# B&R Automation Studio project OpcUaSample410_BrbLibUa103 (part 4)

#### BrbReadDir.c - Gibt eine Liste der Dateien eines Laufwerks zurück
```c
/********************************************************************
 * COPYRIGHT -- Bernecker + Rainer
 ********************************************************************
 * Library: BrbLib
 * File: BrbReadDir.c
 * Author: niedermeierr
 * Created: June 17, 2013
 ********************************************************************
 * Implementation of library BrbLib
 ********************************************************************/

#include <bur/plctypes.h>
#ifdef __cplusplus
	extern "C"
	{
#endif

#include "BrbLib.h"
#include <string.h>
#include <AnsiCFunc.h>

#ifdef __cplusplus
	};
#endif

// NOLINTBEGIN(readability-*, bugprone-easily-swappable-parameters, clang-diagnostic-invalid-utf8, clang-diagnostic-invalid-source-encoding, clang-diagnostic-pointer-arith, clang-diagnostic-strict-prototypes, hicpp-uppercase-literal-suffix, cppcoreguidelines-*, performance-*)

// Eigene Enums und Typen
enum Steps_ENUM
{
	eSTEP_INIT,
	eSTEP_GET_FILTER,
	eSTEP_READ_DIR,
	eSTEP_SORT,
};

// Prototypen
BOOL CallUserFilterFunction(struct BrbReadDir* inst, fiDIR_READ_DATA* pFileInfo);
void SortList(struct BrbReadDir* inst);
INT SortTwoEntries(fiDIR_READ_DATA* pEntry1, fiDIR_READ_DATA* pEntry2, BrbFileSorting_ENUM eSorting, BOOL bCaseSensitive, UDINT pUserCompareFunction);
INT FileComparerNone(fiDIR_READ_DATA* pEntry1, fiDIR_READ_DATA* pEntry2);
INT FileComparerAlphUp(fiDIR_READ_DATA* pEntry1, fiDIR_READ_DATA* pEntry2);
INT FileComparerAlphUpCaseSensitive(fiDIR_READ_DATA* pEntry1, fiDIR_READ_DATA* pEntry2);
INT FileComparerAlphDown(fiDIR_READ_DATA* pEntry1, fiDIR_READ_DATA* pEntry2);
INT FileComparerAlphDownCaseSensitive(fiDIR_READ_DATA* pEntry1, fiDIR_READ_DATA* pEntry2);
INT FileComparerOldest(fiDIR_READ_DATA* pEntry1, fiDIR_READ_DATA* pEntry2);
INT FileComparerYoungest(fiDIR_READ_DATA* pEntry1, fiDIR_READ_DATA* pEntry2);
INT FileComparerBiggest(fiDIR_READ_DATA* pEntry1, fiDIR_READ_DATA* pEntry2);
INT FileComparerSmallest(fiDIR_READ_DATA* pEntry1, fiDIR_READ_DATA* pEntry2);

/* Gibt eine Liste der Dateien und/oder der Verzeichnisse eines Laufwerks zurück */
void BrbReadDir(struct BrbReadDir* inst) // NOLINT(readability-function-cognitive-complexity)
{
	// Prüfung der Parameter
	if(inst->pDevice == 0)
	{
		inst->nStatus = eBRB_ERR_NULL_POINTER;
		return;
	}
	if(inst->pFileFilter == 0)
	{
		inst->nStatus = eBRB_ERR_NULL_POINTER;
		return;
	}

	if(inst->pList == 0)
	{
		inst->nStatus = eBRB_ERR_NULL_POINTER;
		return;
	}

	switch(inst->eStep)
	{
		case eSTEP_INIT:
			// Fub initialisieren
			inst->nStatus = eBRB_ERR_BUSY;
			inst->nDirCount = 0;
			inst->nFileCount = 0;
			inst->nTotalCount = 0;
			memset(&inst->FilterListMan, 0, sizeof(inst->FilterListMan));
			memset(&inst->fbDirRead, 0, sizeof(inst->fbDirRead));
			memset(&inst->FileInfo, 0, sizeof(inst->FileInfo));
			memset(&inst->FileListMan, 0, sizeof(inst->FileListMan));
			// Der Einfachkeit halber wird das File-Array in einer MemList verwaltet
			inst->FileListMan.pList = inst->pList;
			inst->FileListMan.nIndexMax = inst->nListIndexMax;
			inst->FileListMan.nEntryLength = sizeof(inst->ReadListEntry);
			BrbMemListClear(&inst->FileListMan);
			// Prüfen, ob bei benutzerdefinierter Filterung eine Funktion angegeben ist
			inst->eStep = eSTEP_GET_FILTER;
			if(inst->bUserFilter == 1)
			{
				if(inst->pUserFilterFunction == 0)
				{
					inst->nStatus = fiERR_PARAMETER;
					inst->eStep = eSTEP_INIT;
				}
			}
			// Prüfen, ob bei benutzerdefinierter Sortierung eine Vergleichsfunktion angegeben ist
			if(inst->eSorting == eBRB_FILE_SORTING_USER)
			{
				if(inst->pUserCompareFunction == 0)
				{
					inst->nStatus = fiERR_PARAMETER;
					inst->eStep = eSTEP_INIT;
				}
			}
			break;

		case eSTEP_GET_FILTER:
			// Filtertext in Liste umsetzen
			// Der Einfachkeit halber wird die Filter-Liste in einer MemList verwaltet
			inst->FilterListMan.pList = (UDINT)&inst->FilterList;
			inst->FilterListMan.nIndexMax = nBRB_FILTER_SINGLE_INDEX_MAX;
			inst->FilterListMan.nEntryLength = nBRB_FILTER_SINGLE_CHAR_MAX+1;
			BrbMemListClear(&inst->FilterListMan);
			if(strlen(inst->pFileFilter))
			{
				inst->FilterListMan.nEntryCount = BrbStringSplit(inst->pFileFilter, ";", inst->FilterListMan.pList, inst->FilterListMan.nIndexMax, inst->FilterListMan.nEntryLength);
			}
			inst->eStep = eSTEP_READ_DIR;
			break;

		case eSTEP_READ_DIR:
			// Laufwerk auslesen
			inst->nStatus = eBRB_ERR_BUSY;
			inst->fbDirRead.enable = 1;
			inst->fbDirRead.pDevice = (UDINT)inst->pDevice;
			inst->fbDirRead.pPath = (UDINT)inst->pPath;
			inst->fbDirRead.option = fiBOTH;
			inst->fbDirRead.pData = (UDINT)&inst->FileInfo;
			inst->fbDirRead.data_len = sizeof(inst->FileInfo);
			DirRead(&inst->fbDirRead);
			if(inst->fbDirRead.status == 0)
			{
				// Filterprüfung
				BOOL bInFilter = 0;
				// Interner Filter (Dateiendung)
				if((strcmp((STRING*)&inst->FileInfo.Filename, "..") == 0 && inst->bWithParentDir == 0) || strcmp((STRING*)&inst->FileInfo.Filename, ".") == 0)
				{
					// ".." bezieht sich auf das übergeordnete Verzeichnis und wird nur optional zurückgegeben
					// "." bezieht sich auf das eigene Verzeichnis und wird grundsätzlich nicht zurückgegeben
				}
				else if(strcmp((STRING*)&inst->FileInfo.Filename, "..") == 0 && inst->bWithParentDir == 1)
				{
					// ".." bezieht sich auf das übergeordnete Verzeichnis und wird nur optional zurückgegeben
					bInFilter = 1;
					inst->nDirCount += 1;
				}
				else if(inst->eFilter != eBRB_DIR_INFO_ONLY_FILES && inst->FileInfo.Filelength == 0)
				{
					// Verzeichnis
					BOOL bInUserFilter = CallUserFilterFunction(inst, &inst->FileInfo);
					if(bInUserFilter == 1)
					{
						bInFilter = 1;
						inst->nDirCount += 1;
					}
				}
				else if(inst->eFilter != eBRB_DIR_INFO_ONLY_DIRS && inst->FileInfo.Filelength > 0)
				{
					if(inst->FilterListMan.nEntryCount > 0)
					{
						UDINT nFilterListIndex = 0;
						for(nFilterListIndex=0; nFilterListIndex<inst->FilterListMan.nEntryCount; nFilterListIndex++)
						{
							if(BrbStringEndsWith((STRING*)&inst->FileInfo.Filename, inst->FilterList[nFilterListIndex]) == 1)
							{
								// Datei
								BOOL bInUserFilter = CallUserFilterFunction(inst, &inst->FileInfo);
								if(bInUserFilter == 1)
								{
									bInFilter = 1;
									inst->nFileCount += 1;
								}
								break;
							}
						}
					}
					else
					{
						// Datei
						BOOL bInUserFilter = CallUserFilterFunction(inst, &inst->FileInfo);
						if(bInUserFilter == 1)
						{
							bInFilter = 1;
							inst->nFileCount += 1;
						}
					}
				}
				if(bInFilter == 1)
				{
					// Im Filter
					memset(&inst->ReadListEntry, 0, sizeof(inst->ReadListEntry));
					memcpy(&inst->ReadListEntry, &inst->FileInfo, sizeof(inst->ReadListEntry));
					if(inst->FileListMan.nEntryCount <= inst->FileListMan.nIndexMax)
					{
						// Liste ist nicht voll -> in Liste eintragen
						BrbMemListIn(&inst->FileListMan, inst->FileListMan.nEntryCount, (UDINT)&inst->ReadListEntry);
					}
					else
					{
						// Liste ist voll
						// Sortieren
						SortList(inst);
						// Den letzten Eintrag mit dem aktuellen vergleichen
						fiDIR_READ_DATA* pFileInfoLast = (fiDIR_READ_DATA*)(inst->FileListMan.pList + ((inst->FileListMan.nEntryCount-1) * inst->FileListMan.nEntryLength));
						INT nSort = SortTwoEntries(pFileInfoLast, &inst->FileInfo, inst->eSorting, inst->bCaseSensitive, inst->pUserCompareFunction);
						if(nSort > 0)
						{
							// Neue Datei ist näher am Filter als der letzte Eintrag -> ersetzen
							inst->FileListMan.nEntryCount -= 1;
							BrbMemListIn(&inst->FileListMan, inst->FileListMan.nEntryCount, (UDINT)&inst->ReadListEntry);
						}
					}
				}
				memset(&inst->FileInfo, 0, sizeof(inst->FileInfo));
				inst->fbDirRead.entry += 1;
			}
			else if(inst->fbDirRead.status == fiERR_NO_MORE_ENTRIES)
			{
				// Alle Dateien gelesen
				inst->nTotalCount = inst->nDirCount + inst->nFileCount;
				inst->eStep = eSTEP_SORT;
			}
			else if(inst->fbDirRead.status != eBRB_ERR_BUSY)
			{
				inst->nStatus = inst->fbDirRead.status;
				inst->eStep = eSTEP_INIT;
			}
			break;

		case eSTEP_SORT:
			inst->nStatus = eBRB_ERR_BUSY;
			SortList(inst);
			inst->nStatus = eBRB_ERR_OK;
			inst->eStep = eSTEP_INIT;
			break;

	}
}

BOOL CallUserFilterFunction(struct BrbReadDir* inst, fiDIR_READ_DATA* pFileInfo)
{
	BOOL bResult = 0;
	if(inst->bUserFilter == 1)
	{
		if(inst->pUserFilterFunction != 0)
		{
			// Funktion hinterlegt -> Funktionspointer casten
			BOOL (*pFpFunction) (BrbReadDirListEntry_TYP*) = (void*)inst->pUserFilterFunction; // NOLINT(clang-diagnostic-pedantic)
			// Funktion mit Kopie des Eintrags aufrufen
			BrbReadDirListEntry_TYP Entry;
			memset(&Entry, 0, sizeof(Entry));
			memcpy(&Entry, pFileInfo, sizeof(Entry));
			bResult = (*pFpFunction)(&Entry);
		}
	}
	else
	{
		bResult = 1;
	}
	return bResult;
}

void SortList(struct BrbReadDir* inst)
{
	switch(inst->eSorting)
	{
		case eBRB_FILE_SORTING_NONE:
			qsort((fiDIR_READ_DATA*)inst->pList, inst->nListIndexMax+1, sizeof(fiDIR_READ_DATA), (void*)&FileComparerNone); // NOLINT(clang-diagnostic-pedantic
			break;

		case eBRB_FILE_SORTING_ALPH_UP:
			if(inst->bCaseSensitive == 1)
			{
				qsort((fiDIR_READ_DATA*)inst->pList, inst->nListIndexMax+1, sizeof(fiDIR_READ_DATA), (void*)&FileComparerAlphUpCaseSensitive); // NOLINT(clang-diagnostic-pedantic
			}
			else
			{
				qsort((fiDIR_READ_DATA*)inst->pList, inst->nListIndexMax+1, sizeof(fiDIR_READ_DATA), (void*)&FileComparerAlphUp); // NOLINT(clang-diagnostic-pedantic
			}
			break;

		case eBRB_FILE_SORTING_ALPH_DOWN:
			if(inst->bCaseSensitive == 1)
			{
				qsort((fiDIR_READ_DATA*)inst->pList, inst->nListIndexMax+1, sizeof(fiDIR_READ_DATA), (void*)&FileComparerAlphDownCaseSensitive); // NOLINT(clang-diagnostic-pedantic
			}
			else
			{
				qsort((fiDIR_READ_DATA*)inst->pList, inst->nListIndexMax+1, sizeof(fiDIR_READ_DATA), (void*)&FileComparerAlphDown); // NOLINT(clang-diagnostic-pedantic
			}
			break;

		case eBRB_FILE_SORTING_OLDEST:
			qsort((fiDIR_READ_DATA*)inst->pList, inst->nListIndexMax+1, sizeof(fiDIR_READ_DATA), (void*)&FileComparerOldest); // NOLINT(clang-diagnostic-pedantic
			break;

		case eBRB_FILE_SORTING_YOUNGEST:
			qsort((fiDIR_READ_DATA*)inst->pList, inst->nListIndexMax+1, sizeof(fiDIR_READ_DATA), (void*)&FileComparerYoungest); // NOLINT(clang-diagnostic-pedantic
			break;

		case eBRB_FILE_SORTING_BIGGEST:
			qsort((fiDIR_READ_DATA*)inst->pList, inst->nListIndexMax+1, sizeof(fiDIR_READ_DATA), (void*)&FileComparerBiggest); // NOLINT(clang-diagnostic-pedantic
			break;

		case eBRB_FILE_SORTING_SMALLEST:
			qsort((fiDIR_READ_DATA*)inst->pList, inst->nListIndexMax+1, sizeof(fiDIR_READ_DATA), (void*)&FileComparerSmallest); // NOLINT(clang-diagnostic-pedantic
			break;

		case eBRB_FILE_SORTING_USER:
			if(inst->pUserCompareFunction != 0)
			{
				// Funktion hinterlegt -> Funktionspointer übergeben
				qsort((fiDIR_READ_DATA*)inst->pList, inst->nListIndexMax+1, sizeof(BrbReadDirListEntry_TYP), (void*)inst->pUserCompareFunction); // NOLINT(clang-diagnostic-pedantic
			}
			else
			{
				// Funktion nicht hinterlegt -> keine Sortierung
			}
			break;
	}
}

INT SortTwoEntries(fiDIR_READ_DATA* pEntry1, fiDIR_READ_DATA* pEntry2, BrbFileSorting_ENUM eSorting, BOOL bCaseSensitive, UDINT pUserCompareFunction)
{
	INT nResult = 0;
	switch(eSorting) // NOLINT(hicpp-multiway-paths-covered)
	{
		case eBRB_FILE_SORTING_NONE:
			nResult = FileComparerNone(pEntry1, pEntry2);
			break;

		case eBRB_FILE_SORTING_ALPH_UP:
			if(bCaseSensitive == 1)
			{
				nResult = FileComparerAlphUpCaseSensitive(pEntry1, pEntry2);
			}
			else
			{
				nResult = FileComparerAlphUp(pEntry1, pEntry2);
			}
			break;

		case eBRB_FILE_SORTING_ALPH_DOWN:
			if(bCaseSensitive == 1)
			{
				nResult = FileComparerAlphDownCaseSensitive(pEntry1, pEntry2);
			}
			else
			{
				nResult = FileComparerAlphDown(pEntry1, pEntry2);
			}
			break;

		case eBRB_FILE_SORTING_OLDEST:
			nResult = FileComparerOldest(pEntry1, pEntry2);
			break;

		case eBRB_FILE_SORTING_YOUNGEST:
			nResult = FileComparerYoungest(pEntry1, pEntry2);
			break;

		case eBRB_FILE_SORTING_BIGGEST:
			nResult = FileComparerBiggest(pEntry1, pEntry2);
			break;

		case eBRB_FILE_SORTING_SMALLEST:
			nResult = FileComparerSmallest(pEntry1, pEntry2);
			break;

		case eBRB_FILE_SORTING_USER:
			if(pUserCompareFunction != 0)
			{
				// Funktion hinterlegt -> Funktionspointer casten
				INT (*pFpFunction) (BrbReadDirListEntry_TYP*, BrbReadDirListEntry_TYP*) = (void*)pUserCompareFunction; // NOLINT(clang-diagnostic-pedantic)
					// Funktion aufrufen
					nResult = (*pFpFunction)((BrbReadDirListEntry_TYP*) pEntry1, (BrbReadDirListEntry_TYP*)pEntry2);
			}
			else
			{
				// Funktion nicht hinterlegt -> keine Sortierung
				return 0;
			}
			break;

	}
	return nResult;
}

INT FileComparerNone(fiDIR_READ_DATA* pEntry1, fiDIR_READ_DATA* pEntry2)
{
	// Die Verzeichnisse müssen oben sein

	// Anpassung für Compiler-Version V6.3.0: Das Setzen von nResult und Zurückgeben am Ende der Funktion bewirkte, dass die leeren Elemente
	// ganz oben und die gefüllten Elemente ganz unten waren. Jetzt wird der Rückgabewert direkt im If-Block zurückgegeben.
	//INT nResult = 0;

	UDINT nNameLen1 = strlen((STRING*)&pEntry1->Filename);
	UDINT nNameLen2 = strlen((STRING*)&pEntry2->Filename);
	// NOLINTBEGIN(bugprone-branch-clone)
	if(nNameLen1 == 0 && nNameLen2 == 0)
	{
		return (0);
	}
	else if(nNameLen1 == 0)
	{
		return (1);
	}
	else if(nNameLen2 == 0)
	{
		return (-1);
	}
	else if(pEntry1->Filelength == 0 && pEntry2->Filelength > 0)
	{
		return (-1);
	}
	else if(pEntry1->Filelength > 0 && pEntry2->Filelength == 0)
	{
		return (1);
	}
	else if(strcmp((STRING*)&pEntry1->Filename, "..") == 0)
	{
		return (-1);
	}
	else if(strcmp((STRING*)&pEntry2->Filename, "..") == 0)
	{
		return (1);
	}
	else
	{
		return (0);
	}
	// NOLINTEND(bugprone-branch-clone)
}

INT FileComparerAlphUp(fiDIR_READ_DATA* pEntry1, fiDIR_READ_DATA* pEntry2)
{
	UDINT nNameLen1 = strlen((STRING*)&pEntry1->Filename);
	UDINT nNameLen2 = strlen((STRING*)&pEntry2->Filename);
	// NOLINTBEGIN(bugprone-branch-clone)
	if(nNameLen1 == 0 && nNameLen2 == 0)
	{
		return (0);
	}
	else if(nNameLen1 == 0)
	{
		return (1);
	}
	else if(nNameLen2 == 0)
	{
		return (-1);
	}
	else if(pEntry1->Filelength == 0 && pEntry2->Filelength > 0)
	{
		return (-1);
	}
	else if(pEntry1->Filelength > 0 && pEntry2->Filelength == 0)
	{
		return (1);
	}
	else if(strcmp((STRING*)&pEntry1->Filename, "..") == 0)
	{
		return (-1);
	}
	else if(strcmp((STRING*)&pEntry2->Filename, "..") == 0)
	{
		return (1);
	}
	else
	{
		STRING sFilename1[nBRB_FILE_NAME_CHAR_MAX];
		BrbStringCopy(sFilename1, (STRING*)&pEntry1->Filename, sizeof(sFilename1));
		BrbStringToUpper(sFilename1);
		STRING sFilename2[nBRB_FILE_NAME_CHAR_MAX];
		BrbStringCopy(sFilename2, (STRING*)&pEntry2->Filename, sizeof(sFilename2));
		BrbStringToUpper(sFilename2);
		return (INT)(strcmp((STRING*)&sFilename1, (STRING*)&sFilename2));
	}
	// NOLINTEND(bugprone-branch-clone)
}

INT FileComparerAlphUpCaseSensitive(fiDIR_READ_DATA* pEntry1, fiDIR_READ_DATA* pEntry2)
{
	UDINT nNameLen1 = strlen((STRING*)&pEntry1->Filename);
	UDINT nNameLen2 = strlen((STRING*)&pEntry2->Filename);
	// NOLINTBEGIN(bugprone-branch-clone)
	if(nNameLen1 == 0 && nNameLen2 == 0)
	{
		return (0);
	}
	else if(nNameLen1 == 0)
	{
		return (1);
	}
	else if(nNameLen2 == 0)
	{
		return (-1);
	}
	else if(pEntry1->Filelength == 0 && pEntry2->Filelength > 0)
	{
		return (-1);
	}
	else if(pEntry1->Filelength > 0 && pEntry2->Filelength == 0)
	{
		return (1);
	}
	else if(strcmp((STRING*)&pEntry1->Filename, "..") == 0)
	{
		return (-1);
	}
	else if(strcmp((STRING*)&pEntry2->Filename, "..") == 0)
	{
		return (1);
	}
	else
	{
		return (INT)(strcmp((STRING*)&pEntry1->Filename, (STRING*)&pEntry2->Filename));
	}
	// NOLINTEND(bugprone-branch-clone)
}

INT FileComparerAlphDown(fiDIR_READ_DATA* pEntry1, fiDIR_READ_DATA* pEntry2)
{
	UDINT nNameLen1 = strlen((STRING*)&pEntry1->Filename);
	UDINT nNameLen2 = strlen((STRING*)&pEntry2->Filename);
	// NOLINTBEGIN(bugprone-branch-clone)
	if(nNameLen1 == 0 && nNameLen2 == 0)
	{
		return (0);
	}
	else if(nNameLen1 == 0)
	{
		return (1);
	}
	else if(nNameLen2 == 0)
	{
		return (-1);
	}
	else if(pEntry1->Filelength == 0 && pEntry2->Filelength > 0)
	{
		return (-1);
	}
	else if(pEntry1->Filelength > 0 && pEntry2->Filelength == 0)
	{
		return (1);
	}
	else if(strcmp((STRING*)&pEntry1->Filename, "..") == 0)
	{
		return (-1);
	}
	else if(strcmp((STRING*)&pEntry2->Filename, "..") == 0)
	{
		return (1);
	}
	else
	{
		STRING sFilename1[nBRB_FILE_NAME_CHAR_MAX];
		BrbStringCopy(sFilename1, (STRING*)&pEntry1->Filename, sizeof(sFilename1));
		BrbStringToUpper(sFilename1);
		STRING sFilename2[nBRB_FILE_NAME_CHAR_MAX];
		BrbStringCopy(sFilename2, (STRING*)&pEntry2->Filename, sizeof(sFilename2));
		BrbStringToUpper(sFilename2);
		return (INT)(strcmp((STRING*)&sFilename2, (STRING*)&sFilename1));
	}
	// NOLINTEND(bugprone-branch-clone)
}

INT FileComparerAlphDownCaseSensitive(fiDIR_READ_DATA* pEntry1, fiDIR_READ_DATA* pEntry2)
{
	UDINT nNameLen1 = strlen((STRING*)&pEntry1->Filename);
	UDINT nNameLen2 = strlen((STRING*)&pEntry2->Filename);
	// NOLINTBEGIN(bugprone-branch-clone)
	if(nNameLen1 == 0 && nNameLen2 == 0)
	{
		return (0);
	}
	else if(nNameLen1 == 0)
	{
		return (1);
	}
	else if(nNameLen2 == 0)
	{
		return (-1);
	}
	else if(pEntry1->Filelength == 0 && pEntry2->Filelength > 0)
	{
		return (-1);
	}
	else if(pEntry1->Filelength > 0 && pEntry2->Filelength == 0)
	{
		return (1);
	}
	else if(strcmp((STRING*)&pEntry1->Filename, "..") == 0)
	{
		return (-1);
	}
	else if(strcmp((STRING*)&pEntry2->Filename, "..") == 0)
	{
		return (1);
	}
	else
	{
		return (INT)(strcmp((STRING*)&pEntry2->Filename, (STRING*)&pEntry1->Filename));
	}
	// NOLINTEND(bugprone-branch-clone)
}

INT FileComparerOldest(fiDIR_READ_DATA* pEntry1, fiDIR_READ_DATA* pEntry2)
{
	UDINT nNameLen1 = strlen((STRING*)&pEntry1->Filename);
	UDINT nNameLen2 = strlen((STRING*)&pEntry2->Filename);
	// NOLINTBEGIN(bugprone-branch-clone)
	if(nNameLen1 == 0 && nNameLen2 == 0)
	{
		return (0);
	}
	else if(nNameLen1 == 0)
	{
		return (1);
	}
	else if(nNameLen2 == 0)
	{
		return (-1);
	}
	else if(pEntry1->Filelength == 0 && pEntry2->Filelength > 0)
	{
		return (-1);
	}
	else if(pEntry1->Filelength > 0 && pEntry2->Filelength == 0)
	{
		return (1);
	}
	else if(strcmp((STRING*)&pEntry1->Filename, "..") == 0)
	{
		return (-1);
	}
	else if(strcmp((STRING*)&pEntry2->Filename, "..") == 0)
	{
		return (1);
	}
	else
	{
		if(pEntry1->Date < pEntry2->Date)
		{
			return (-1);
		}
		else if(pEntry1->Date > pEntry2->Date)
		{
			return (1);
		}
		else
		{
			return (FileComparerAlphUp(pEntry1, pEntry2));
		}
	}
	// NOLINTEND(bugprone-branch-clone)
}

INT FileComparerYoungest(fiDIR_READ_DATA* pEntry1, fiDIR_READ_DATA* pEntry2)
{
	UDINT nNameLen1 = strlen((STRING*)&pEntry1->Filename);
	UDINT nNameLen2 = strlen((STRING*)&pEntry2->Filename);
	// NOLINTBEGIN(bugprone-branch-clone)
	if(nNameLen1 == 0 && nNameLen2 == 0)
	{
		return (0);
	}
	else if(nNameLen1 == 0)
	{
		return (1);
	}
	else if(nNameLen2 == 0)
	{
		return (-1);
	}
	else if(pEntry1->Filelength == 0 && pEntry2->Filelength > 0)
	{
		return (-1);
	}
	else if(pEntry1->Filelength > 0 && pEntry2->Filelength == 0)
	{
		return (1);
	}
	else if(strcmp((STRING*)&pEntry1->Filename, "..") == 0)
	{
		return (-1);
	}
	else if(strcmp((STRING*)&pEntry2->Filename, "..") == 0)
	{
		return (1);
	}
	else
	{
		if(pEntry1->Date > pEntry2->Date)
		{
			return (-1);
		}
		else if(pEntry1->Date < pEntry2->Date)
		{
			return (1);
		}
		else
		{
			return (FileComparerAlphUp(pEntry1, pEntry2));
		}
	}
	// NOLINTEND(bugprone-branch-clone)
}

INT FileComparerBiggest(fiDIR_READ_DATA* pEntry1, fiDIR_READ_DATA* pEntry2)
{
	UDINT nNameLen1 = strlen((STRING*)&pEntry1->Filename);
	UDINT nNameLen2 = strlen((STRING*)&pEntry2->Filename);
	// NOLINTBEGIN(bugprone-branch-clone)
	if(nNameLen1 == 0 && nNameLen2 == 0)
	{
		return (0);
	}
	else if(nNameLen1 == 0)
	{
		return (1);
	}
	else if(nNameLen2 == 0)
	{
		return (-1);
	}
	else if(pEntry1->Filelength == 0 && pEntry2->Filelength > 0)
	{
		return (-1);
	}
	else if(pEntry1->Filelength > 0 && pEntry2->Filelength == 0)
	{
		return (1);
	}
	else if(strcmp((STRING*)&pEntry1->Filename, "..") == 0)
	{
		return (-1);
	}
	else if(strcmp((STRING*)&pEntry2->Filename, "..") == 0)
	{
		return (1);
	}
	else
	{
		if(pEntry1->Filelength > pEntry2->Filelength)
		{
			return (-1);
		}
		else if(pEntry1->Filelength < pEntry2->Filelength)
		{
			return (1);
		}
		else
		{
			return (FileComparerAlphUp(pEntry1, pEntry2));
		}
	}
	// NOLINTEND(bugprone-branch-clone)
}

INT FileComparerSmallest(fiDIR_READ_DATA* pEntry1, fiDIR_READ_DATA* pEntry2)
{
	UDINT nNameLen1 = strlen((STRING*)&pEntry1->Filename);
	UDINT nNameLen2 = strlen((STRING*)&pEntry2->Filename);
	// NOLINTBEGIN(bugprone-branch-clone)
	if(nNameLen1 == 0 && nNameLen2 == 0)
	{
		return (0);
	}
	else if(nNameLen1 == 0)
	{
		return (1);
	}
	else if(nNameLen2 == 0)
	{
		return (-1);
	}
	else if(pEntry1->Filelength == 0 && pEntry2->Filelength > 0)
	{
		return (-1);
	}
	else if(pEntry1->Filelength > 0 && pEntry2->Filelength == 0)
	{
		return (1);
	}
	else if(strcmp((STRING*)&pEntry1->Filename, "..") == 0)
	{
		return (-1);
	}
	else if(strcmp((STRING*)&pEntry2->Filename, "..") == 0)
	{
		return (1);
	}
	else
	{
		if(pEntry1->Filelength < pEntry2->Filelength)
		{
			return (-1);
		}
		else if(pEntry1->Filelength > pEntry2->Filelength)
		{
			return (1);
		}
		else
		{
			return (FileComparerAlphUp(pEntry1, pEntry2));
		}
	}
	// NOLINTEND(bugprone-branch-clone)
}

// NOLINTEND(readability-*, bugprone-easily-swappable-parameters, clang-diagnostic-invalid-utf8, clang-diagnostic-invalid-source-encoding, clang-diagnostic-pointer-arith, clang-diagnostic-strict-prototypes, hicpp-uppercase-literal-suffix, cppcoreguidelines-*, performance-*)
```

#### BrbDeleteFiles.c - Löscht Dateien, die älter als das angegebene Datum sind
```c
/********************************************************************
 * COPYRIGHT -- Bernecker + Rainer
 ********************************************************************
 * Library: BrbLib
 * File: BrbDeleteFiles.c
 * Author: niedermeierr
 * Created: January 26, 2015
 ********************************************************************
 * Implementation of library BrbLib
 ********************************************************************/

#include <bur/plctypes.h>
#ifdef __cplusplus
	extern "C"
	{
#endif

	#include "BrbLib.h"
	#include <string.h>
	#include <AnsiCFunc.h>

#ifdef __cplusplus
	};
#endif

// NOLINTBEGIN(readability-*, bugprone-easily-swappable-parameters, clang-diagnostic-invalid-utf8, clang-diagnostic-invalid-source-encoding, clang-diagnostic-pointer-arith, clang-diagnostic-strict-prototypes, hicpp-uppercase-literal-suffix, cppcoreguidelines-*, performance-*)

// Eigene Enums und Typen
enum Steps_ENUM
{
	eSTEP_INIT,
	eSTEP_GET_FILTER,
	eSTEP_READ_DIR,
	eSTEP_DELETE_FILE,
};

/* Löscht Dateien, die über Filter festgelegt sind */
void BrbDeleteFiles(struct BrbDeleteFiles* inst) // NOLINT(readability-function-cognitive-complexity)
{
	// Prüfung der Parameter
	if(inst->pDevice == 0)
	{
		inst->nStatus = eBRB_ERR_NULL_POINTER;
		return;
	}
	if(inst->pFileFilter == 0)
	{
		inst->nStatus = eBRB_ERR_NULL_POINTER;
		return;
	}

	switch(inst->eStep)
	{
		case eSTEP_INIT:
			// Fub initialisieren
			inst->nStatus = eBRB_ERR_BUSY;
			inst->nDeletedFileCount = 0;
			inst->nKeptFileCount = 0;
			memset(&inst->FilterListMan, 0, sizeof(inst->FilterListMan));
			memset(&inst->fbDirRead, 0, sizeof(inst->fbDirRead));
			memset(&inst->FileInfo, 0, sizeof(inst->FileInfo));
			inst->eStep = eSTEP_GET_FILTER;
			break;

		case eSTEP_GET_FILTER:
			// Filtertext in Liste umsetzen
			// Der Einfachkeit halber wird die Filter-Liste in einer MemList verwaltet
			inst->FilterListMan.pList = (UDINT)&inst->FilterList;
			inst->FilterListMan.nIndexMax = nBRB_FILTER_SINGLE_INDEX_MAX;
			inst->FilterListMan.nEntryLength = nBRB_FILTER_SINGLE_CHAR_MAX+1;
			BrbMemListClear(&inst->FilterListMan);
			if(strlen(inst->pFileFilter))
			{
				inst->FilterListMan.nEntryCount = BrbStringSplit(inst->pFileFilter, ";", inst->FilterListMan.pList, inst->FilterListMan.nIndexMax, inst->FilterListMan.nEntryLength);
			}
			inst->eStep = eSTEP_READ_DIR;
			break;

		case eSTEP_READ_DIR:
			// Laufwerk auslesen
			inst->nStatus = eBRB_ERR_BUSY;
			inst->fbDirRead.enable = 1;
			inst->fbDirRead.pDevice = (UDINT)inst->pDevice;
			inst->fbDirRead.pPath = (UDINT)inst->pPath;
			inst->fbDirRead.option = fiFILE;
			inst->fbDirRead.pData = (UDINT)&inst->FileInfo;
			inst->fbDirRead.data_len = sizeof(inst->FileInfo);
			DirRead(&inst->fbDirRead);
			if(inst->fbDirRead.status == 0)
			{
				BOOL bInFilter = 0;
				// Datumsprüfung
				if(inst->FileInfo.Date >= inst->dtDateStart && inst->FileInfo.Date <= inst->dtDateEnd)
				{
					// Filterprüfung
					if(inst->FilterListMan.nEntryCount > 0)
					{
						UDINT nFilterListIndex = 0;
						for(nFilterListIndex=0; nFilterListIndex<inst->FilterListMan.nEntryCount; nFilterListIndex++)
						{
							if(BrbStringEndsWith((STRING*)&inst->FileInfo.Filename, inst->FilterList[nFilterListIndex]) == 1)
							{
								// Datei
								bInFilter = 1;
								break;
							}
						}
					}
					else
					{
						bInFilter = 1;
					}
				}
				if(bInFilter == 1)
				{
					// Datei löschen
					memset(&inst->fbFileDelete, 0, sizeof(inst->fbFileDelete));
					memset(&inst->sFileWithPath, 0, sizeof(inst->sFileWithPath));
					if(inst->pPath != 0)
					{
						BrbCombinePath((STRING*)inst->pPath, (STRING*)&inst->FileInfo.Filename, (STRING*)&inst->sFileWithPath);
					}
					else
					{
						BrbStringCat((STRING*)&inst->sFileWithPath, (STRING*)&inst->FileInfo.Filename, sizeof(inst->sFileWithPath));
					}
					inst->nDeletedFileCount += 1;
					inst->eStep = eSTEP_DELETE_FILE;
				}
				else
				{
					inst->nKeptFileCount += 1;
					inst->fbDirRead.entry += 1;
				}
				memset(&inst->FileInfo, 0, sizeof(inst->FileInfo));
			}
			else if(inst->fbDirRead.status == fiERR_NO_MORE_ENTRIES)
			{
				// Alle Dateien gelesen -> Fertig
				inst->nStatus = 0;
				inst->eStep = eSTEP_INIT;
			}
			else if(inst->fbDirRead.status != eBRB_ERR_BUSY)
			{
				inst->nStatus = inst->fbDirRead.status;
				inst->eStep = eSTEP_INIT;
			}
			break;

		case eSTEP_DELETE_FILE:
			inst->nStatus = eBRB_ERR_BUSY;
			inst->fbFileDelete.enable = 1;
			inst->fbFileDelete.pDevice = (UDINT)inst->pDevice;
			inst->fbFileDelete.pName = (UDINT)&inst->sFileWithPath;
			FileDelete(&inst->fbFileDelete);
			if(inst->fbFileDelete.status == 0)
			{
				inst->eStep = eSTEP_READ_DIR;
			}
			else if(inst->fbFileDelete.status != eBRB_ERR_BUSY)
			{
				inst->nStatus = inst->fbFileDelete.status;
				inst->eStep = eSTEP_INIT;
			}
			break;

	}
}

// NOLINTEND(readability-*, bugprone-easily-swappable-parameters, clang-diagnostic-invalid-utf8, clang-diagnostic-invalid-source-encoding, clang-diagnostic-pointer-arith, clang-diagnostic-strict-prototypes, hicpp-uppercase-literal-suffix, cppcoreguidelines-*, performance-*)
```

#### BrbLoadFileDataObj.c - Lädt eine Datei in ein Datenobjekt
```c
/********************************************************************
 * COPYRIGHT -- Bernecker + Rainer
 ********************************************************************
 * Library: BrbLib
 * File: BrbLoadFileDataObj.c
 * Author: niedermeierr
 * Created: June 25, 2013
 ********************************************************************
 * Implementation of library BrbLib
 ********************************************************************/

#include <bur/plctypes.h>
#ifdef __cplusplus
	extern "C"
	{
#endif

#include "BrbLib.h"
#include <string.h>
#include <AnsiCFunc.h>

#ifdef __cplusplus
	};
#endif

// NOLINTBEGIN(readability-*, bugprone-easily-swappable-parameters, clang-diagnostic-invalid-utf8, clang-diagnostic-invalid-source-encoding, clang-diagnostic-pointer-arith, clang-diagnostic-strict-prototypes, hicpp-uppercase-literal-suffix, cppcoreguidelines-*, performance-*)

// Eigene Enums und Typen
enum Steps_ENUM
{
	eSTEP_INIT,
	eSTEP_GET_DAT_OBJ,
	eSTEP_DEL_DATA_OBJ,
	eSTEP_OPEN_FILE,
	eSTEP_CREATE_DAT_OBJ,
	eSTEP_READ_FILE,
	eSTEP_CLOSE_FILE,
	eSTEP_ERR_CLOSE_FILE,
	eSTEP_ERR_DEL_DATA_OBJ,
};

/* Lädt eine Datei in ein Datenobjekt */
void BrbLoadFileDataObj(struct BrbLoadFileDataObj* inst) // NOLINT(readability-function-cognitive-complexity)
{
	// Prüfung der Parameter
	if(inst->pDevice == 0)
	{
		inst->nStatus = eBRB_ERR_NULL_POINTER;
		return;
	}
	if(inst->pFile == 0)
	{
		inst->nStatus = eBRB_ERR_NULL_POINTER;
		return;
	}
	if(inst->pDataObjName == 0)
	{
		inst->nStatus = eBRB_ERR_NULL_POINTER;
		return;
	}

	switch(inst->eStep)
	{
		case eSTEP_INIT:
			// Fub initialisieren
			inst->nStatus = inst->nStatusIntern = eBRB_ERR_BUSY;
			inst->nDataObjIdent = 0;
			inst->pDataObjMem = 0;
			inst->nDataObjLen = 0;
			memset(&inst->fbDatObjInfo, 0, sizeof(inst->fbDatObjInfo));
			memset(&inst->fbDatObjDelete, 0, sizeof(inst->fbDatObjDelete));
			memset(&inst->fbFileOpen, 0, sizeof(inst->fbFileOpen));
			memset(&inst->fbDatObjCreate, 0, sizeof(inst->fbDatObjCreate));
			memset(&inst->fbFileRead, 0, sizeof(inst->fbFileRead));
			memset(&inst->fbFileClose, 0, sizeof(inst->fbFileClose));
			inst->eStep = eSTEP_GET_DAT_OBJ;
			break;

		case eSTEP_GET_DAT_OBJ:
			// Evtl. unter diesem Namen schon vorhandenes Datenobjekt finden
			inst->nStatus = inst->nStatusIntern = eBRB_ERR_BUSY;
			inst->fbDatObjInfo.enable = 1;
			inst->fbDatObjInfo.pName = (UDINT)inst->pDataObjName;
			DatObjInfo(&inst->fbDatObjInfo);
			if(inst->fbDatObjInfo.status == 0)
			{
				inst->eStep = eSTEP_DEL_DATA_OBJ;
			}
			else if(inst->fbDatObjInfo.status != eBRB_ERR_BUSY)
			{
				inst->eStep = eSTEP_OPEN_FILE;
			}
			break;

		case eSTEP_DEL_DATA_OBJ:
			// Evtl. unter diesem Namen schon vorhandenes Datenobjekt löschen
			inst->nStatus = inst->nStatusIntern = eBRB_ERR_BUSY;
			inst->fbDatObjDelete.enable = 1;
			inst->fbDatObjDelete.ident = inst->fbDatObjInfo.ident;
			DatObjDelete(&inst->fbDatObjDelete);
			if(inst->fbDatObjDelete.status != eBRB_ERR_BUSY)
			{
				inst->eStep = eSTEP_OPEN_FILE;
			}
			break;

		case eSTEP_OPEN_FILE:
			// Datei öffnen
			inst->nStatus = inst->nStatusIntern = eBRB_ERR_BUSY;
			inst->fbFileOpen.enable = 1;
			inst->fbFileOpen.pDevice = (UDINT)inst->pDevice;
			inst->fbFileOpen.pFile = (UDINT)inst->pFile;
			inst->fbFileOpen.mode = fiREAD_ONLY;
			FileOpen(&inst->fbFileOpen);
			if(inst->fbFileOpen.status == 0)
			{
				inst->eStep = eSTEP_CREATE_DAT_OBJ;
			}
			else if(inst->fbFileOpen.status != eBRB_ERR_BUSY)
			{
				inst->nStatus = inst->nStatusIntern = inst->fbFileOpen.status;
				inst->nDataObjIdent = 0;
				inst->pDataObjMem = 0;
				inst->nDataObjLen = 0;
				inst->eStep = eSTEP_INIT;
			}
			break;

		case eSTEP_CREATE_DAT_OBJ:
			// Datenobjekt von der Größe der Datei erzeugen
			inst->nStatus = inst->nStatusIntern = eBRB_ERR_BUSY;
			inst->fbDatObjCreate.enable = 1;
			inst->fbDatObjCreate.grp = 0;
			inst->fbDatObjCreate.pName = (UDINT)inst->pDataObjName;
			inst->fbDatObjCreate.len = inst->fbFileOpen.filelen;
			inst->fbDatObjCreate.MemType = inst->nDataObjMemType;
			inst->fbDatObjCreate.Option = inst->nDataObjOption;
			inst->fbDatObjCreate.pCpyData = 0;
			DatObjCreate(&inst->fbDatObjCreate);
			if(inst->fbDatObjCreate.status == 0)
			{
				memset((USINT*)inst->fbDatObjCreate.pDatObjMem, 0, inst->fbDatObjCreate.len);
				inst->nDataObjIdent = inst->fbDatObjCreate.ident;
				inst->pDataObjMem = inst->fbDatObjCreate.pDatObjMem;
				inst->nDataObjLen = inst->fbDatObjCreate.len;
				inst->eStep = eSTEP_READ_FILE;
			}
			else if(inst->fbDatObjCreate.status != eBRB_ERR_BUSY)
			{
				inst->nStatusIntern = inst->fbDatObjCreate.status;
				inst->eStep = eSTEP_ERR_CLOSE_FILE;
			}
			break;

		case eSTEP_READ_FILE:
			// Datei in das Datenpbjekt lesen
			inst->nStatus = inst->nStatusIntern = eBRB_ERR_BUSY;
			inst->fbFileRead.enable = 1;
			inst->fbFileRead.ident = inst->fbFileOpen.ident;
			inst->fbFileRead.offset = 0;
			inst->fbFileRead.pDest = inst->fbDatObjCreate.pDatObjMem;
			inst->fbFileRead.len = inst->fbDatObjCreate.len;
			FileRead(&inst->fbFileRead);
			if(inst->fbFileRead.status == 0)
			{
				inst->eStep = eSTEP_CLOSE_FILE;
			}
			else if(inst->fbFileRead.status != eBRB_ERR_BUSY)
			{
				inst->nStatusIntern = inst->fbFileRead.status;
				inst->eStep = eSTEP_ERR_CLOSE_FILE;
			}
			break;

		case eSTEP_CLOSE_FILE:
			// Datei schliessen
			inst->nStatus = inst->nStatusIntern = eBRB_ERR_BUSY;
			inst->fbFileClose.enable = 1;
			inst->fbFileClose.ident = inst->fbFileOpen.ident;
			FileClose(&inst->fbFileClose);
			if(inst->fbFileClose.status == 0)
			{
				inst->nStatus = inst->nStatusIntern = 0;
				inst->eStep = eSTEP_INIT;
			}
			else if(inst->fbFileClose.status != eBRB_ERR_BUSY)
			{
				inst->nStatusIntern = inst->fbFileClose.status;
				inst->eStep = eSTEP_ERR_DEL_DATA_OBJ;
			}
			break;

		case eSTEP_ERR_CLOSE_FILE:
			// Datei im Fehlerfall schliessen
			inst->nStatus = eBRB_ERR_BUSY;
			inst->fbFileClose.enable = 1;
			inst->fbFileClose.ident = inst->fbFileOpen.ident;
			FileClose(&inst->fbFileClose);
			if(inst->fbFileClose.status != eBRB_ERR_BUSY)
			{
				if(inst->fbDatObjCreate.ident != 0)
				{
					inst->eStep = eSTEP_ERR_DEL_DATA_OBJ;
				}
				else
				{
					inst->nStatus = inst->nStatusIntern;
					inst->nDataObjIdent = 0;
					inst->pDataObjMem = 0;
					inst->nDataObjLen = 0;
					inst->eStep = eSTEP_INIT;
				}
			}
			break;

		case eSTEP_ERR_DEL_DATA_OBJ:
			// Datenobjekt im Fehlerfall löschen
			inst->nStatus = eBRB_ERR_BUSY;
			inst->fbDatObjDelete.enable = 1;
			inst->fbDatObjDelete.ident = inst->fbDatObjInfo.ident;
			DatObjDelete(&inst->fbDatObjDelete);
			if(inst->fbDatObjDelete.status != eBRB_ERR_BUSY)
			{
				inst->nStatus = inst->nStatusIntern;
				inst->nDataObjIdent = 0;
				inst->pDataObjMem = 0;
				inst->nDataObjLen = 0;
				inst->eStep = eSTEP_INIT;
			}
			break;

	}
}

// NOLINTEND(readability-*, bugprone-easily-swappable-parameters, clang-diagnostic-invalid-utf8, clang-diagnostic-invalid-source-encoding, clang-diagnostic-pointer-arith, clang-diagnostic-strict-prototypes, hicpp-uppercase-literal-suffix, cppcoreguidelines-*, performance-*)
```

#### BrbSaveFileDataObj.c - Speichert ein Datenobjekt in eine Datei
```c
/********************************************************************
 * COPYRIGHT -- Bernecker + Rainer
 ********************************************************************
 * Library: BrbLib
 * File: BrbSaveFileDataObj.c
 * Author: niedermeierr
 * Created: June 25, 2013
 ********************************************************************
 * Implementation of library BrbLib
 ********************************************************************/

#include <bur/plctypes.h>
#ifdef __cplusplus
	extern "C"
	{
#endif

#include "BrbLib.h"
#include <string.h>
#include <AnsiCFunc.h>

#ifdef __cplusplus
	};
#endif

// NOLINTBEGIN(readability-*, bugprone-easily-swappable-parameters, clang-diagnostic-invalid-utf8, clang-diagnostic-invalid-source-encoding, clang-diagnostic-pointer-arith, clang-diagnostic-strict-prototypes, hicpp-uppercase-literal-suffix, cppcoreguidelines-*, performance-*)

// Eigene Enums und Typen
enum Steps_ENUM
{
	eSTEP_INIT,
	eSTEP_GET_DAT_OBJ,
	eSTEP_GET_FILE,
	eSTEP_DEL_FILE,
	eSTEP_CREATE_FILE,
	eSTEP_WRITE_FILE,
	eSTEP_CLOSE_FILE,
	eSTEP_ERR_CLOSE_FILE,
};

/* Speichert ein Datenobjekt in eine Datei */
void BrbSaveFileDataObj(struct BrbSaveFileDataObj* inst)
{
	// Prüfung der Parameter
	if(inst->pDevice == 0)
	{
		inst->nStatus = eBRB_ERR_NULL_POINTER;
		return;
	}
	if(inst->pFile == 0)
	{
		inst->nStatus = eBRB_ERR_NULL_POINTER;
		return;
	}
	if(inst->pDataObjName == 0)
	{
		inst->nStatus = eBRB_ERR_NULL_POINTER;
		return;
	}

	switch(inst->eStep)
	{
		case eSTEP_INIT:
			// Fub initialisieren
			inst->nStatus = inst->nStatusIntern = eBRB_ERR_BUSY;
			memset(&inst->fbDatObjInfo, 0, sizeof(inst->fbDatObjInfo));
			memset(&inst->fbFileInfo, 0, sizeof(inst->fbFileInfo));
			memset(&inst->fbFileDelete, 0, sizeof(inst->fbFileDelete));
			memset(&inst->fbFileCreate, 0, sizeof(inst->fbFileCreate));
			memset(&inst->fbFileWrite, 0, sizeof(inst->fbFileWrite));
			memset(&inst->fbFileClose, 0, sizeof(inst->fbFileClose));
			inst->eStep = eSTEP_GET_DAT_OBJ;
			break;

		case eSTEP_GET_DAT_OBJ:
			// Prüfen, ob es das angegebene Datenobjekt gibt
			inst->nStatus = inst->nStatusIntern = eBRB_ERR_BUSY;
			inst->fbDatObjInfo.enable = 1;
			inst->fbDatObjInfo.pName = (UDINT)inst->pDataObjName;
			DatObjInfo(&inst->fbDatObjInfo);
			if(inst->fbDatObjInfo.status == 0)
			{
				inst->eStep = eSTEP_GET_FILE;
			}
			else if(inst->fbDatObjInfo.status != eBRB_ERR_BUSY)
			{
				inst->nStatus = inst->nStatusIntern = inst->fbDatObjInfo.status;
				inst->eStep = eSTEP_INIT;
			}
			break;

		case eSTEP_GET_FILE:
			// Prüfen, ob es die Datei schon gibt
			inst->nStatus = inst->nStatusIntern = eBRB_ERR_BUSY;
			inst->fbFileInfo.enable = 1;
			inst->fbFileInfo.pDevice = (UDINT)inst->pDevice;
			inst->fbFileInfo.pName = (UDINT)inst->pFile;
			inst->fbFileInfo.pInfo = (UDINT)&inst->FileInfo;
			FileInfo(&inst->fbFileInfo);
			if(inst->fbFileInfo.status == 0)
			{
				inst->eStep = eSTEP_DEL_FILE;
			}
			else if(inst->fbFileInfo.status != eBRB_ERR_BUSY)
			{
				inst->eStep = eSTEP_CREATE_FILE;
			}
			break;

		case eSTEP_DEL_FILE:
			// Evtl. schon vorhandene Datei löschen
			inst->nStatus = inst->nStatusIntern = eBRB_ERR_BUSY;
			inst->fbFileDelete.enable = 1;
			inst->fbFileDelete.pDevice = (UDINT)inst->pDevice;
			inst->fbFileDelete.pName = (UDINT)inst->pFile;
			FileDelete(&inst->fbFileDelete);
			if(inst->fbFileDelete.status != eBRB_ERR_BUSY)
			{
				inst->eStep = eSTEP_CREATE_FILE;
			}
			break;

		case eSTEP_CREATE_FILE:
			// Datei erzeugen
			inst->nStatus = inst->nStatusIntern = eBRB_ERR_BUSY;
			inst->fbFileCreate.enable = 1;
			inst->fbFileCreate.pDevice = (UDINT)inst->pDevice;
			inst->fbFileCreate.pFile = (UDINT)inst->pFile;
			FileCreate(&inst->fbFileCreate);
			if(inst->fbFileCreate.status == 0)
			{
				inst->eStep = eSTEP_WRITE_FILE;
			}
			else if(inst->fbFileCreate.status != eBRB_ERR_BUSY)
			{
				inst->nStatus = inst->nStatusIntern = inst->fbFileCreate.status;
				inst->eStep = eSTEP_INIT;
			}
			break;

		case eSTEP_WRITE_FILE:
			// Datenobjekt in die Datei schreiben
			inst->nStatus = inst->nStatusIntern = eBRB_ERR_BUSY;
			inst->fbFileWrite.enable = 1;
			inst->fbFileWrite.ident = inst->fbFileCreate.ident;
			inst->fbFileWrite.offset = 0;
			inst->fbFileWrite.pSrc = inst->fbDatObjInfo.pDatObjMem;
			inst->fbFileWrite.len = inst->fbDatObjInfo.len;
			FileWrite(&inst->fbFileWrite);
			if(inst->fbFileWrite.status == 0)
			{
				inst->eStep = eSTEP_CLOSE_FILE;
			}
			else if(inst->fbFileWrite.status != eBRB_ERR_BUSY)
			{
				inst->nStatusIntern = inst->fbFileWrite.status;
				inst->eStep = eSTEP_ERR_CLOSE_FILE;
			}
			break;

		case eSTEP_CLOSE_FILE:
			// Datei schliessen
			inst->nStatus = inst->nStatusIntern = eBRB_ERR_BUSY;
			inst->fbFileClose.enable = 1;
			inst->fbFileClose.ident = inst->fbFileCreate.ident;
			FileClose(&inst->fbFileClose);
			if(inst->fbFileClose.status == 0)
			{
				inst->nStatus = inst->nStatusIntern = 0;
				inst->eStep = eSTEP_INIT;
			}
			else if(inst->fbFileClose.status != eBRB_ERR_BUSY)
			{
				inst->nStatus = inst->nStatusIntern = inst->fbFileClose.status;
				inst->eStep = eSTEP_INIT;
			}
			break;

		case eSTEP_ERR_CLOSE_FILE:
			// Datei im Fehlerfall schliessen
			inst->nStatus = eBRB_ERR_BUSY;
			inst->fbFileClose.enable = 1;
			inst->fbFileClose.ident = inst->fbFileCreate.ident;
			FileClose(&inst->fbFileClose);
			if(inst->fbFileClose.status != eBRB_ERR_BUSY)
			{
				inst->nStatus = inst->nStatusIntern;
				inst->eStep = eSTEP_INIT;
			}
			break;

	}
}

// NOLINTEND(readability-*, bugprone-easily-swappable-parameters, clang-diagnostic-invalid-utf8, clang-diagnostic-invalid-source-encoding, clang-diagnostic-pointer-arith, clang-diagnostic-strict-prototypes, hicpp-uppercase-literal-suffix, cppcoreguidelines-*, performance-*)
```

#### BrbLoadFileBin.c - Lädt eine binäre Datei in ein Byte-Array
```c
#include <bur/plctypes.h>
#ifdef __cplusplus
	extern "C"
	{
#endif

	#include "BrbLib.h"
	#include <string.h>
	#include <AnsiCFunc.h>

#ifdef __cplusplus
	};
#endif

// NOLINTBEGIN(readability-*, bugprone-easily-swappable-parameters, clang-diagnostic-invalid-utf8, clang-diagnostic-invalid-source-encoding, clang-diagnostic-pointer-arith, clang-diagnostic-strict-prototypes, hicpp-uppercase-literal-suffix, cppcoreguidelines-*, performance-*)

// Eigene Enums und Typen
enum Steps_ENUM
{
	eSTEP_INIT,
	eSTEP_OPEN_FILE,
	eSTEP_CHECK_SIZE,
	eSTEP_READ_FILE,
	eSTEP_CLOSE_FILE,
	eSTEP_ERR_CLOSE_FILE,
};

/* Lädt eine Datei in eine Feld-Variable */
void BrbLoadFileBin(struct BrbLoadFileBin* inst)
{
	// Prüfung der Parameter
	if(inst->pDevice == 0)
	{
		inst->nStatus = eBRB_ERR_NULL_POINTER;
		return;
	}
	if(inst->pFile == 0)
	{
		inst->nStatus = eBRB_ERR_NULL_POINTER;
		return;
	}
	if(inst->pVar == 0)
	{
		inst->nStatus = eBRB_ERR_NULL_POINTER;
		return;
	}

	switch(inst->eStep)
	{
		case eSTEP_INIT:
			// Fub initialisieren
			inst->nStatus = inst->nStatusIntern = eBRB_ERR_BUSY;
			memset((USINT*)inst->pVar, 0, inst->nVarSize);
			inst->nValidBytes = 0;
			memset(&inst->fbFileOpen, 0, sizeof(inst->fbFileOpen));
			memset(&inst->fbFileReadEx, 0, sizeof(inst->fbFileReadEx));
			memset(&inst->fbFileClose, 0, sizeof(inst->fbFileClose));
			inst->eStep = eSTEP_OPEN_FILE;
			break;

		case eSTEP_OPEN_FILE:
			// Datei öffnen
			inst->nStatus = inst->nStatusIntern = eBRB_ERR_BUSY;
			inst->fbFileOpen.enable = 1;
			inst->fbFileOpen.pDevice = (UDINT)inst->pDevice;
			inst->fbFileOpen.pFile = (UDINT)inst->pFile;
			inst->fbFileOpen.mode = fiREAD_ONLY;
			FileOpen(&inst->fbFileOpen);
			if(inst->fbFileOpen.status == 0)
			{
				inst->eStep = eSTEP_CHECK_SIZE;
			}
			else if(inst->fbFileOpen.status != eBRB_ERR_BUSY)
			{
				inst->nStatus = inst->nStatusIntern = inst->fbFileOpen.status;
				inst->eStep = eSTEP_INIT;
			}
			break;

		case eSTEP_CHECK_SIZE:
			// Datei- und Variablen-Größe prüfen
			if(inst->nVarSize >= inst->fbFileOpen.filelen)
			{
				inst->eStep = eSTEP_READ_FILE;
			}
			else
			{
				inst->nStatusIntern = fiERR_DATA_SIZE; // = 20701
				inst->eStep = eSTEP_ERR_CLOSE_FILE;
			}
			break;

		case eSTEP_READ_FILE:
			// Datei in das Datenpbjekt lesen
			inst->nStatus = inst->nStatusIntern = eBRB_ERR_BUSY;
			inst->fbFileReadEx.enable = 1;
			inst->fbFileReadEx.ident = inst->fbFileOpen.ident;
			inst->fbFileReadEx.offset = 0;
			inst->fbFileReadEx.pDest = (UDINT)inst->pVar;
			inst->fbFileReadEx.len = inst->fbFileOpen.filelen;
			FileReadEx(&inst->fbFileReadEx);
			if(inst->fbFileReadEx.status == 0)
			{
				inst->nValidBytes = inst->fbFileReadEx.bytesread;
				inst->eStep = eSTEP_CLOSE_FILE;
			}
			else if(inst->fbFileReadEx.status != eBRB_ERR_BUSY)
			{
				inst->nStatusIntern = inst->fbFileReadEx.status;
				inst->eStep = eSTEP_ERR_CLOSE_FILE;
			}
			break;

		case eSTEP_CLOSE_FILE:
			// Datei schliessen
			inst->nStatus = inst->nStatusIntern = eBRB_ERR_BUSY;
			inst->fbFileClose.enable = 1;
			inst->fbFileClose.ident = inst->fbFileOpen.ident;
			FileClose(&inst->fbFileClose);
			if(inst->fbFileClose.status == 0)
			{
				inst->nStatus = inst->nStatusIntern = 0;
				inst->eStep = eSTEP_INIT;
			}
			else if(inst->fbFileClose.status != eBRB_ERR_BUSY)
			{
				inst->nStatusIntern = inst->fbFileClose.status;
				inst->eStep = eSTEP_INIT;
			}
			break;

		case eSTEP_ERR_CLOSE_FILE:
			// Datei im Fehlerfall schliessen
			inst->nStatus = eBRB_ERR_BUSY;
			inst->fbFileClose.enable = 1;
			inst->fbFileClose.ident = inst->fbFileOpen.ident;
			FileClose(&inst->fbFileClose);
			if(inst->fbFileClose.status != eBRB_ERR_BUSY)
			{
				inst->nStatus = inst->nStatusIntern;
				inst->eStep = eSTEP_INIT;
			}
			break;

	}
}

// NOLINTEND(readability-*, bugprone-easily-swappable-parameters, clang-diagnostic-invalid-utf8, clang-diagnostic-invalid-source-encoding, clang-diagnostic-pointer-arith, clang-diagnostic-strict-prototypes, hicpp-uppercase-literal-suffix, cppcoreguidelines-*, performance-*)
```

#### BrbCheckFileName.c - Ersetzt Sonderzeichen in einem Dateinamen mit Unterstrichen
```c
/********************************************************************
 * COPYRIGHT -- Bernecker + Rainer
 ********************************************************************
 * Library: BrbLib
 * File: BrbCheckFileName.c
 * Author: niedermeierr
 * Created: July 25, 2013
 ********************************************************************
 * Implementation of library BrbLib
 ********************************************************************/

#include <bur/plctypes.h>
#ifdef __cplusplus
	extern "C"
	{
#endif

#include "BrbLib.h"
#include <string.h>

#ifdef __cplusplus
	};
#endif

// NOLINTBEGIN(readability-*, bugprone-easily-swappable-parameters, clang-diagnostic-invalid-utf8, clang-diagnostic-invalid-source-encoding, clang-diagnostic-pointer-arith, clang-diagnostic-strict-prototypes, hicpp-uppercase-literal-suffix, cppcoreguidelines-*, performance-*)

/* Ersetzt Sonderzeichen in einem Datei-Namen mit Unterstrichen */
unsigned short BrbCheckFileName(plcstring* pFileName)
{
	// Prüfung der Parameter
	if(pFileName == 0)
	{
		return eBRB_ERR_NULL_POINTER;
	}
	// Check
	UINT nResult = 0;
	UDINT nLen = strlen(pFileName);
	DINT nCharIndex = 0;
	USINT* pChar = 0;
	UINT nDotCount = 0;
	// Text von hinten nach vorne durchsuchen
	for(nCharIndex=(DINT)nLen-1; nCharIndex>=0; nCharIndex--)
	{
		pChar = (USINT*)(pFileName + nCharIndex);
		if(*pChar == 46)
		{
			// Alle Punkte außer dem letzten werden ersetzt
			nDotCount += 1;
			if(nDotCount > 1)
			{
				*pChar = 95;
				nResult += 1;
			}
		}
		//										-									0 							9									A								Z									_									a								z
		else if(!((*pChar == 45) || (*pChar >= 48 && *pChar <= 57) || (*pChar >= 65 && *pChar <= 90) || (*pChar == 95) || (*pChar >= 97 && *pChar <= 122)))
		{
			// Sonderzeichen werden ersetzt
			*pChar = 95;
			nResult += 1;
		}
	}
	return nResult;
}

// NOLINTEND(readability-*, bugprone-easily-swappable-parameters, clang-diagnostic-invalid-utf8, clang-diagnostic-invalid-source-encoding, clang-diagnostic-pointer-arith, clang-diagnostic-strict-prototypes, hicpp-uppercase-literal-suffix, cppcoreguidelines-*, performance-*)
```

#### BrbCheckFileEnding.c - Prüft die Endung eines Dateinamens und hängt sie gegebenenfalls an
```c
/********************************************************************
 * COPYRIGHT -- Bernecker + Rainer
 ********************************************************************
 * Library: BrbLib
 * File: BrbCheckFileEnding.c
 * Author: niedermeierr
 * Created: July 26, 2013
 ********************************************************************
 * Implementation of library BrbLib
 ********************************************************************/

#include <bur/plctypes.h>
#ifdef __cplusplus
	extern "C"
	{
#endif

#include "BrbLib.h"
#include <string.h>

#ifdef __cplusplus
	};
#endif

// NOLINTBEGIN(readability-*, bugprone-easily-swappable-parameters, clang-diagnostic-invalid-utf8, clang-diagnostic-invalid-source-encoding, clang-diagnostic-pointer-arith, clang-diagnostic-strict-prototypes, hicpp-uppercase-literal-suffix, cppcoreguidelines-*, performance-*)

/* Prüft die Endung eines Datei-Namens und berichtigt sie gegebenenfalls */
plcbit BrbCheckFileEnding(plcstring* pFileName, plcstring* pEnding)
{
	// Prüfung der Parameter
	if(pFileName == 0)
	{
		return 0;
	}
	if(pEnding == 0)
	{
		return 0;
	}
	// Check
	BOOL bResult = 0;
	if(BrbStringEndsWith(pFileName, pEnding) == 0)
	{
		STRING* pFileNameDotAdr = BrbStringGetAdrOf(pFileName, ".", 0);
		if(pFileNameDotAdr != 0)
		{
			// Wegschneiden der vorhandenen Endung
			STRING sFileNameWithoutEnding[nBRB_FILE_NAME_CHAR_MAX];
			BrbStringGetSubTextByAdr(pFileName, pFileNameDotAdr, sFileNameWithoutEnding);
			strcpy(pFileName, sFileNameWithoutEnding); // NOLINT(clang-analyzer-security.insecureAPI.strcpy)
		}
		STRING* pEndingDotAdr = BrbStringGetAdrOf(pEnding, ".", 0);
		if(pEndingDotAdr != 0)
		{
			// Endung beinhaltet den Punkt schon
			strcat(pFileName, pEnding); // NOLINT(clang-analyzer-security.insecureAPI.strcpy)
		}
		else
		{
			// Endung beinhaltet den Punkt noch nicht
			strcat(pFileName, "."); // NOLINT(clang-analyzer-security.insecureAPI.strcpy)
			strcat(pFileName, pEnding); // NOLINT(clang-analyzer-security.insecureAPI.strcpy)
		}
		bResult = 1;
	}
	return bResult;
}

// NOLINTEND(readability-*, bugprone-easily-swappable-parameters, clang-diagnostic-invalid-utf8, clang-diagnostic-invalid-source-encoding, clang-diagnostic-pointer-arith, clang-diagnostic-strict-prototypes, hicpp-uppercase-literal-suffix, cppcoreguidelines-*, performance-*)
```

#### BrbCombinePath.c - Fügt zwei Pfade oder eine Pfad und eine Datei zusammen
```c
/********************************************************************
 * COPYRIGHT -- Bernecker + Rainer
 ********************************************************************
 * Library: BrbLib
 * File: BrbCombinePath.c
 * Author: niedermeierr
 * Created: November 02, 2014
 ********************************************************************
 * Implementation of library BrbLib
 ********************************************************************/

#include <bur/plctypes.h>
#ifdef __cplusplus
	extern "C"
	{
#endif

#include "BrbLib.h"
#include <string.h>

#ifdef __cplusplus
	};
#endif

// NOLINTBEGIN(readability-*, bugprone-easily-swappable-parameters, clang-diagnostic-invalid-utf8, clang-diagnostic-invalid-source-encoding, clang-diagnostic-pointer-arith, clang-diagnostic-strict-prototypes, hicpp-uppercase-literal-suffix, cppcoreguidelines-*, performance-*)

/* Fügt zwei Pfade oder einen Pfad und eine Datei-Namen zusammen */
unsigned short BrbCombinePath(plcstring* pPath, plcstring* pFilename, plcstring* pFilenameWithPath)
{
	// Prüfung der Parameter
	if(pPath == 0)
	{
		return eBRB_ERR_NULL_POINTER;
	}
	if(pFilename == 0)
	{
		return eBRB_ERR_NULL_POINTER;
	}
	if(pFilenameWithPath == 0)
	{
		return eBRB_ERR_NULL_POINTER;
	}
	// Check
	STRING sFileWithPath[nBRB_FILE_NAME_CHAR_MAX];
	memset(sFileWithPath, 0, sizeof(sFileWithPath));
	if(strlen(pPath) > 0)
	{
		BrbStringCat(sFileWithPath, pPath, sizeof(sFileWithPath));
		if(BrbStringEndsWith(pPath, "\\") == 0)
		{
			BrbStringCat(sFileWithPath, "\\", sizeof(sFileWithPath));
		}
	}
	BrbStringCat(sFileWithPath, pFilename, sizeof(sFileWithPath));
	strcpy(pFilenameWithPath, sFileWithPath); // NOLINT(clang-analyzer-security.insecureAPI.strcpy)
	return 0;
}

// NOLINTEND(readability-*, bugprone-easily-swappable-parameters, clang-diagnostic-invalid-utf8, clang-diagnostic-invalid-source-encoding, clang-diagnostic-pointer-arith, clang-diagnostic-strict-prototypes, hicpp-uppercase-literal-suffix, cppcoreguidelines-*, performance-*)
```

#### Package Logical/Libraries/BrbLib/Logger - Logbuch-Funktionen

#### BrbLoggerReadHierarchicalList.c - Durchsucht eine Logbuch
```c
#include <bur/plctypes.h>
#ifdef __cplusplus
	extern "C"
	{
#endif
	#include "BrbLib.h"
#ifdef __cplusplus
	};
#endif

#include <string.h>

// NOLINTBEGIN(readability-*, bugprone-easily-swappable-parameters, clang-diagnostic-invalid-utf8, clang-diagnostic-invalid-source-encoding, clang-diagnostic-pointer-arith, clang-diagnostic-strict-prototypes, hicpp-uppercase-literal-suffix, cppcoreguidelines-*, performance-*)

// Eigene Enums und Typen
enum Steps_ENUM
{
	eSTEP_INIT,
	eSTEP_GET_LOGBOOK,
	eSTEP_CHECK_STARTRECORDID,
	eSTEP_GET_LATEST_RECORDID,
	eSTEP_GET_PREVIOUS_RECORDID,
	eSTEP_READ_RECORD,
	eSTEP_READ_ERRORNUMBER,
	eSTEP_READ_OBJECTID,
	eSTEP_READ_DESCRIPTION,
	eSTEP_INSERT_LIST_ENTRY,
};

/* Liest die zu einem definierten Logger-Eintrag gehörende Hierarchie-Liste von Einträgen aus */
void BrbLoggerReadHierarchicalList(struct BrbLoggerReadHierarchicalList* inst) // NOLINT(readability-function-cognitive-complexity)
{
	switch(inst->eStep)
	{
		case eSTEP_INIT:
			// Fub initialisieren
			inst->nStatus = eBRB_ERR_BUSY;
			memset((USINT*)&inst->ActEntry, 0, sizeof(inst->ActEntry));
			inst->LogListManagement.pList = inst->pLogList;
			inst->LogListManagement.nEntryLength = sizeof(BrbLogHierarchListEntry_TYP);
			inst->LogListManagement.nIndexMax = inst->nLogListIndexMax;
			BrbMemListClear(&inst->LogListManagement);
			inst->nSearchEntryCount = 0;
			inst->bFirstEntryIsListed = 0;
			inst->nListEntryCount = 0;
			// Prüfen, ob LogbookIdent ermittelt werden muss
			if(inst->nEventLogIdent != 0)
			{
				if(strlen(inst->sLogbookName) > 0 && strcmp(inst->sLogbookName, inst->sLastLogbookName) == 0)
				{
					// Gleiches Logbuch wie beim letzten Aufruf
					inst->eStep = eSTEP_CHECK_STARTRECORDID;
				}
				else
				{
					// Logbuch-Name hat sich geändert
					inst->eStep = eSTEP_GET_LOGBOOK;
				}
			}
			else
			{
				// Logbuch wurde noch nicht ermittelt
				inst->eStep = eSTEP_GET_LOGBOOK;
			}
			break;

		case eSTEP_GET_LOGBOOK:
			// Ident des Logbuchs ermitteln
			inst->fbArEventLogGetIdent.Execute = 1;
			BrbStringCopy(inst->fbArEventLogGetIdent.Name, inst->sLogbookName, sizeof(inst->fbArEventLogGetIdent.Name));
			ArEventLogGetIdent(&inst->fbArEventLogGetIdent);
			if(inst->fbArEventLogGetIdent.Done == 1)
			{
				BrbStringCopy(inst->sLastLogbookName, inst->sLogbookName, sizeof(inst->sLastLogbookName));
				inst->nEventLogIdent = inst->fbArEventLogGetIdent.Ident;
				inst->fbArEventLogGetIdent.Execute = 0;
				ArEventLogGetIdent(&inst->fbArEventLogGetIdent);
				inst->eStep = eSTEP_CHECK_STARTRECORDID;
			}
			else if(inst->fbArEventLogGetIdent.Error == 1)
			{
				inst->nEventLogIdent = 0;
				inst->nStatus = inst->fbArEventLogGetIdent.StatusID;
				inst->fbArEventLogGetIdent.Execute = 0;
				ArEventLogGetIdent(&inst->fbArEventLogGetIdent);
				inst->eStep = eSTEP_INIT;
			}
			break;

		case eSTEP_CHECK_STARTRECORDID:
			// Prüfen, ob eine StartRecordId angegeben ist
			if(inst->nStartRecordId != 0)
			{
				inst->ActEntry.nRecordId = inst->nStartRecordId;
				inst->eStep = eSTEP_READ_OBJECTID;
			}
			else
			{
				// Bei jüngstem Eintrag beginnen
				inst->eStep = eSTEP_GET_LATEST_RECORDID;
			}
			break;

		case eSTEP_GET_LATEST_RECORDID:
			// RecordId des jüngsten Eintrag ermitteln
			inst->fbArEventLogGetLatestRecordID.Execute = 1;
			inst->fbArEventLogGetLatestRecordID.Ident = inst->nEventLogIdent;
			ArEventLogGetLatestRecordID(&inst->fbArEventLogGetLatestRecordID);
			if(inst->fbArEventLogGetLatestRecordID.Done == 1)
			{
				inst->ActEntry.nRecordId = inst->fbArEventLogGetLatestRecordID.RecordID;
				inst->fbArEventLogGetLatestRecordID.Execute = 0;
				ArEventLogGetLatestRecordID(&inst->fbArEventLogGetLatestRecordID);
				inst->eStep = eSTEP_READ_OBJECTID;
			}
			else if(inst->fbArEventLogGetLatestRecordID.Error == 1)
			{
				memset((USINT*)&inst->ActEntry, 0, sizeof(inst->ActEntry));
				inst->nStatus = inst->fbArEventLogGetLatestRecordID.StatusID;
				inst->fbArEventLogGetLatestRecordID.Execute = 0;
				ArEventLogGetLatestRecordID(&inst->fbArEventLogGetLatestRecordID);
				inst->eStep = eSTEP_INIT;
			}
			break;

		case eSTEP_GET_PREVIOUS_RECORDID:
			// RecordId des chronologisch vorherigen Eintrags ermitteln
			inst->fbArEventLogGetPreviousRecordID.Execute = 1;
			inst->fbArEventLogGetPreviousRecordID.Ident = inst->nEventLogIdent;
			inst->fbArEventLogGetPreviousRecordID.RecordID = inst->ActEntry.nRecordId;
			ArEventLogGetPreviousRecordID(&inst->fbArEventLogGetPreviousRecordID);
			if(inst->fbArEventLogGetPreviousRecordID.Done == 1)
			{
				inst->ActEntry.nRecordId = inst->fbArEventLogGetPreviousRecordID.PrevRecordID;
				inst->fbArEventLogGetPreviousRecordID.Execute = 0;
				ArEventLogGetPreviousRecordID(&inst->fbArEventLogGetPreviousRecordID);
				inst->eStep = eSTEP_READ_OBJECTID;
			}
			else if(inst->fbArEventLogGetPreviousRecordID.Error == 1)
			{
				memset((USINT*)&inst->ActEntry, 0, sizeof(inst->ActEntry));
				if(inst->fbArEventLogGetPreviousRecordID.StatusID == arEVENTLOG_ERR_RECORDID_INVALID)
				{
					// Am Ende des Logbuchs angekommen
					inst->nStatus = 0;
				}
				else
				{
					inst->nStatus = inst->fbArEventLogGetPreviousRecordID.StatusID;
				}
				inst->fbArEventLogGetPreviousRecordID.Execute = 0;
				ArEventLogGetPreviousRecordID(&inst->fbArEventLogGetPreviousRecordID);
				inst->eStep = eSTEP_INIT;
			}
			break;

		case eSTEP_READ_OBJECTID:
			// Limit prüfen
			if(inst->bFirstEntryIsListed == 0 && (inst->nSearchEntryCountLimit > 0 && inst->nSearchEntryCount > inst->nSearchEntryCountLimit))
			{
				// Limit erreicht -> Ende
				inst->nStatus = 0;
				inst->eStep = eSTEP_INIT;
			}
			else
			{
				// ObjectId ('Entered by') lesen
				inst->fbArEventLogReadObjectID.Execute = 1;
				inst->fbArEventLogReadObjectID.Ident = inst->nEventLogIdent;
				inst->fbArEventLogReadObjectID.RecordID = inst->ActEntry.nRecordId;
				ArEventLogReadObjectID(&inst->fbArEventLogReadObjectID);
				if(inst->fbArEventLogReadObjectID.Done == 1)
				{
					inst->nSearchEntryCount += 1;
					strncpy(inst->ActEntry.sObjectId, inst->fbArEventLogReadObjectID.ObjectID, sizeof(inst->ActEntry.sObjectId));
					inst->fbArEventLogReadObjectID.Execute = 0;
					ArEventLogReadObjectID(&inst->fbArEventLogReadObjectID);
					// ObjectId filtern
					// NOLINTBEGIN(bugprone-branch-clone)
					if(strlen(inst->sObjectId) == 0)
					{
						// Kein Filter
						inst->eStep = eSTEP_READ_RECORD;
					}
					else if(strcmp(inst->sObjectId, inst->ActEntry.sObjectId) == 0)
					{
						inst->eStep = eSTEP_READ_RECORD;
					}
					else
					{
						if(inst->bFirstEntryIsListed == 0)
						{
							// Nächsten Eintrag lesen
							inst->ActEntry.nOriginRecordId = 0;
							inst->ActEntry.nEventId = 0;
							inst->ActEntry.nSeverity = 0;
							memset(inst->ActEntry.sObjectId, 0, sizeof(inst->ActEntry.sObjectId));
							inst->eStep = eSTEP_GET_PREVIOUS_RECORDID;
						}
						else
						{
							// Alle passenden Einträge schon gelistet -> Ende
							inst->nStatus = 0;
							inst->eStep = eSTEP_INIT;
						}
					}
					// NOLINTEND(bugprone-branch-clone)
				}
				else if(inst->fbArEventLogReadObjectID.Error == 1)
				{
					memset((USINT*)&inst->ActEntry, 0, sizeof(inst->ActEntry));
					inst->nStatus = inst->fbArEventLogReadObjectID.StatusID;
					inst->fbArEventLogReadObjectID.Execute = 0;
					ArEventLogReadObjectID(&inst->fbArEventLogReadObjectID);
					inst->eStep = eSTEP_INIT;
				}
			}
			break;

		case eSTEP_READ_RECORD:
			// Logbuch-Eintrag lesen
			inst->fbArEventLogRead.Execute = 1;
			inst->fbArEventLogRead.Ident = inst->nEventLogIdent;
			inst->fbArEventLogRead.RecordID = inst->ActEntry.nRecordId;
			ArEventLogRead(&inst->fbArEventLogRead);
			if(inst->fbArEventLogRead.Done == 1)
			{
				inst->ActEntry.nOriginRecordId = inst->fbArEventLogRead.OriginRecordID;
				inst->ActEntry.nEventId = inst->fbArEventLogRead.EventID;
				UDINT nSeverityMasked = (UDINT)inst->ActEntry.nEventId & 3221225472UL; // =0xC0000000 = Bit30..31 // NOLINT(hicpp-signed-bitwise)
				inst->ActEntry.nSeverity = (USINT)(nSeverityMasked>>30); // NOLINT(hicpp-signed-bitwise)
				inst->fbArEventLogRead.Execute = 0;
				ArEventLogRead(&inst->fbArEventLogRead);
				if(inst->ActEntry.nEventId == 0)
				{
					// Eintrag im ErrorNumber-Format
					inst->ActEntry.nEventId = 0;
					inst->ActEntry.nSeverity = 0;
					inst->eStep = eSTEP_READ_ERRORNUMBER;
				}
				else
				{
					// Eintrag im EventID-Format
					// EventId filtern
					if(inst->nStartEventId == 0 || inst->ActEntry.nEventId == inst->nStartEventId || inst->bFirstEntryIsListed == 1)
					{
						// Severity filtern
						BOOL bInFilter = 0;
						// NOLINTBEGIN(bugprone-branch-clone)
						if(inst->eSeverities == eBRB_LOG_SEVERITY_FILTER_ALL)
						{
							bInFilter = 1;
						}
						else if(((inst->eSeverities & eBRB_LOG_SEVERITY_FILTER_SUCCESS) == eBRB_LOG_SEVERITY_FILTER_SUCCESS) && inst->ActEntry.nSeverity == arEVENTLOG_SEVERITY_SUCCESS) // NOLINT(hicpp-signed-bitwise)
						{
							bInFilter = 1;
						}
						else if(((inst->eSeverities & eBRB_LOG_SEVERITY_FILTER_INFO) == eBRB_LOG_SEVERITY_FILTER_INFO) && inst->ActEntry.nSeverity == arEVENTLOG_SEVERITY_INFO) // NOLINT(hicpp-signed-bitwise)
						{
							bInFilter = 1;
						}
						else if(((inst->eSeverities & eBRB_LOG_SEVERITY_FILTER_WARNING) == eBRB_LOG_SEVERITY_FILTER_WARNING) && inst->ActEntry.nSeverity == arEVENTLOG_SEVERITY_WARNING) // NOLINT(hicpp-signed-bitwise)
						{
							bInFilter = 1;
						}
						else if(((inst->eSeverities & eBRB_LOG_SEVERITY_FILTER_ERROR) == eBRB_LOG_SEVERITY_FILTER_ERROR) && inst->ActEntry.nSeverity == arEVENTLOG_SEVERITY_ERROR) // NOLINT(hicpp-signed-bitwise)
						{
							bInFilter = 1;
						}
						if(bInFilter == 1)
						{
							inst->eStep = eSTEP_READ_DESCRIPTION;
						}
						else
						{
							if(inst->bFirstEntryIsListed == 0)
							{
								// Nächsten Eintrag lesen
								inst->ActEntry.nOriginRecordId = 0;
								inst->ActEntry.nEventId = 0;
								inst->ActEntry.nSeverity = 0;
								inst->eStep = eSTEP_GET_PREVIOUS_RECORDID;
							}
							else
							{
								// Alle passenden Einträge schon gelistet -> Ende
								inst->nStatus = 0;
								inst->eStep = eSTEP_INIT;
							}
						}
						// NOLINTEND(bugprone-branch-clone)
					}
					else
					{
						// Nächsten Eintrag lesen
						inst->ActEntry.nOriginRecordId = 0;
						inst->ActEntry.nEventId = 0;
						inst->ActEntry.nSeverity = 0;
						inst->eStep = eSTEP_GET_PREVIOUS_RECORDID;
					}
				}
			}
			else if(inst->fbArEventLogRead.Error == 1)
			{
				memset((USINT*)&inst->ActEntry, 0, sizeof(inst->ActEntry));
				inst->nStatus = inst->fbArEventLogRead.StatusID;
				inst->fbArEventLogRead.Execute = 0;
				ArEventLogRead(&inst->fbArEventLogRead);
				inst->eStep = eSTEP_INIT;
			}
			break;

		case eSTEP_READ_ERRORNUMBER:
			// Fehlernummer und Severity eines alten Eintrags lesen
			inst->fbArEventLogReadErrorNumber.Execute = 1;
			inst->fbArEventLogReadErrorNumber.Ident = inst->nEventLogIdent;
			inst->fbArEventLogReadErrorNumber.RecordID = inst->ActEntry.nRecordId;
			ArEventLogReadErrorNumber(&inst->fbArEventLogReadErrorNumber);
			if(inst->fbArEventLogReadErrorNumber.Done == 1)
			{
				inst->ActEntry.nEventId = (DINT)inst->fbArEventLogReadErrorNumber.ErrorNumber;
				inst->ActEntry.nSeverity = inst->fbArEventLogReadErrorNumber.Severity;
				inst->fbArEventLogReadErrorNumber.Execute = 0;
				ArEventLogReadErrorNumber(&inst->fbArEventLogReadErrorNumber);
				// ErrorNumber filtern
				if(inst->nStartEventId == 0 || inst->ActEntry.nEventId == inst->nStartEventId || inst->bFirstEntryIsListed == 1)
				{
					// Severity filtern
					BOOL bInFilter = 0;
					// NOLINTBEGIN(bugprone-branch-clone)
					if(inst->eSeverities == eBRB_LOG_SEVERITY_FILTER_ALL)
					{
						bInFilter = 1;
					}
					else if(((inst->eSeverities & eBRB_LOG_SEVERITY_FILTER_SUCCESS) == eBRB_LOG_SEVERITY_FILTER_SUCCESS) && inst->ActEntry.nSeverity == arEVENTLOG_SEVERITY_SUCCESS) // NOLINT(hicpp-signed-bitwise)
					{
						bInFilter = 1;
					}
					else if(((inst->eSeverities & eBRB_LOG_SEVERITY_FILTER_INFO) == eBRB_LOG_SEVERITY_FILTER_INFO) && inst->ActEntry.nSeverity == arEVENTLOG_SEVERITY_INFO) // NOLINT(hicpp-signed-bitwise)
					{
						bInFilter = 1;
					}
					else if(((inst->eSeverities & eBRB_LOG_SEVERITY_FILTER_WARNING) == eBRB_LOG_SEVERITY_FILTER_WARNING) && inst->ActEntry.nSeverity == arEVENTLOG_SEVERITY_WARNING) // NOLINT(hicpp-signed-bitwise)
					{
						bInFilter = 1;
					}
					else if(((inst->eSeverities & eBRB_LOG_SEVERITY_FILTER_ERROR) == eBRB_LOG_SEVERITY_FILTER_ERROR) && inst->ActEntry.nSeverity == arEVENTLOG_SEVERITY_ERROR) // NOLINT(hicpp-signed-bitwise)
					{
						bInFilter = 1;
					}
					// NOLINTEND(bugprone-branch-clone)
					if(bInFilter == 1)
					{
						inst->eStep = eSTEP_READ_DESCRIPTION;
					}
					else
					{
						if(inst->bFirstEntryIsListed == 0)
						{
							// Nächsten Eintrag lesen
							inst->ActEntry.nOriginRecordId = 0;
							inst->ActEntry.nEventId = 0;
							inst->ActEntry.nSeverity = 0;
							inst->eStep = eSTEP_GET_PREVIOUS_RECORDID;
						}
						else
						{
							// Alle passenden Einträge schon gelistet -> Ende
							inst->nStatus = 0;
							inst->eStep = eSTEP_INIT;
						}
					}
				}
				else
				{
					// Nächsten Eintrag lesen
					inst->ActEntry.nOriginRecordId = 0;
					inst->ActEntry.nEventId = 0;
					inst->ActEntry.nSeverity = 0;
					inst->eStep = eSTEP_GET_PREVIOUS_RECORDID;
				}
			}
			else if(inst->fbArEventLogReadErrorNumber.Error == 1)
			{
				memset((USINT*)&inst->ActEntry, 0, sizeof(inst->ActEntry));
				inst->nStatus = inst->fbArEventLogReadErrorNumber.StatusID;
				inst->fbArEventLogReadErrorNumber.Execute = 0;
				ArEventLogReadErrorNumber(&inst->fbArEventLogReadErrorNumber);
				inst->eStep = eSTEP_INIT;
			}
			break;

		case eSTEP_READ_DESCRIPTION:
			// Description lesen
			inst->fbArEventLogReadDescription.Execute = 1;
			inst->fbArEventLogReadDescription.Ident = inst->nEventLogIdent;
			inst->fbArEventLogReadDescription.RecordID = inst->ActEntry.nRecordId;
			BrbStringCopy(inst->fbArEventLogReadDescription.LanguageCode, inst->sLanguageCode, sizeof(inst->fbArEventLogReadDescription.LanguageCode));
			inst->fbArEventLogReadDescription.TextBuffer = (UDINT)&inst->ActEntry.sDecription;
			inst->fbArEventLogReadDescription.TextBufferSize = sizeof(inst->ActEntry.sDecription);
			ArEventLogReadDescription(&inst->fbArEventLogReadDescription);
			if(inst->fbArEventLogReadDescription.Done == 1)
			{
				inst->fbArEventLogReadDescription.Execute = 0;
				ArEventLogReadDescription(&inst->fbArEventLogReadDescription);
				inst->eStep = eSTEP_INSERT_LIST_ENTRY;
			}
			else if(inst->fbArEventLogReadDescription.Error == 1)
			{
				memset((USINT*)&inst->ActEntry, 0, sizeof(inst->ActEntry));
				inst->nStatus = inst->fbArEventLogReadDescription.StatusID;
				inst->fbArEventLogReadDescription.Execute = 0;
				ArEventLogReadDescription(&inst->fbArEventLogReadDescription);
				inst->eStep = eSTEP_INIT;
			}
			break;

		case eSTEP_INSERT_LIST_ENTRY:
			// Einfügen des Eintrags in die Liste
			BrbMemListIn(&inst->LogListManagement, 0, (UDINT)&inst->ActEntry);
			inst->nListEntryCount = (UINT)inst->LogListManagement.nEntryCount;
			inst->bFirstEntryIsListed = 1;
			if(inst->ActEntry.nOriginRecordId != 0)
			{
				// Nächsten hierarchischen Eintrag lesen
				ArEventLogRecordIDType nOriginRecordId = inst->ActEntry.nOriginRecordId;
				memset((USINT*)&inst->ActEntry, 0, sizeof(inst->ActEntry));
				inst->ActEntry.nRecordId = nOriginRecordId;
				inst->eStep = eSTEP_READ_OBJECTID;
			}
			else
			{
				// Kein weiterer hierachischer Eintrag -> Ende
				inst->nStatus = 0;
				inst->eStep = eSTEP_INIT;
			}
			break;

	}
}

// NOLINTEND(readability-*, bugprone-easily-swappable-parameters, clang-diagnostic-invalid-utf8, clang-diagnostic-invalid-source-encoding, clang-diagnostic-pointer-arith, clang-diagnostic-strict-prototypes, hicpp-uppercase-literal-suffix, cppcoreguidelines-*, performance-*)
```

#### Package Logical/Libraries/BrbLib/TimeAndDate - Zeit- und Datums-Funktionen

#### BrbSetDtStruct.c - Setzt eine DTStructure
```c
/********************************************************************
 * COPYRIGHT -- Bernecker + Rainer
 ********************************************************************
 * Library: BrbLib
 * File: BrbSetDtStruct.c
 * Author: niedermeierr
 * Created: May 18, 2021
 ********************************************************************
 * Implementation of library BrbLib
 ********************************************************************/

#include <bur/plctypes.h>
#ifdef __cplusplus
	extern "C"
	{
#endif

#include "BrbLib.h"
#include "AsTime.h" // NOLINT(clang-diagnostic-nonportable-system-include-path)

#ifdef __cplusplus
	};
#endif

// NOLINTBEGIN(readability-*, bugprone-easily-swappable-parameters, clang-diagnostic-invalid-utf8, clang-diagnostic-invalid-source-encoding, clang-diagnostic-pointer-arith, clang-diagnostic-strict-prototypes, hicpp-uppercase-literal-suffix, cppcoreguidelines-*, performance-*)

/* Setzt eine DTStructure-Zeit */
plcdt BrbSetDtStruct(struct DTStructure* pDtStruct, unsigned short nYear, unsigned char nMonth, unsigned char nDay, unsigned char nHour, unsigned char nMinute, unsigned char nSecond, unsigned short nMillisecond, unsigned short nMicrosecond)
{
	pDtStruct->year = nYear;
	pDtStruct->month = nMonth;
	pDtStruct->day = nDay;
	pDtStruct->hour = nHour;
	pDtStruct->minute = nMinute;
	pDtStruct->second = nSecond;
	pDtStruct->millisec = nMillisecond;
	pDtStruct->microsec =  nMicrosecond;
	BrbGetWeekdayDtStruct(pDtStruct);
	return DTStructure_TO_DT((UDINT)pDtStruct);
}

// NOLINTEND(readability-*, bugprone-easily-swappable-parameters, clang-diagnostic-invalid-utf8, clang-diagnostic-invalid-source-encoding, clang-diagnostic-pointer-arith, clang-diagnostic-strict-prototypes, hicpp-uppercase-literal-suffix, cppcoreguidelines-*, performance-*)
```

#### BrbSetDt.c - Setzt eine DATE_AND_TIME-Angabe
```c
/********************************************************************
 * COPYRIGHT -- Bernecker + Rainer
 ********************************************************************
 * Library: BrbLib
 * File: BrbSetDtStruct.c
 * Author: niedermeierr
 * Created: May 18, 2021
 ********************************************************************
 * Implementation of library BrbLib
 ********************************************************************/

#include <bur/plctypes.h>
#ifdef __cplusplus
	extern "C"
	{
#endif

#include "BrbLib.h"
#include "AsTime.h" // NOLINT(clang-diagnostic-nonportable-system-include-path)

#ifdef __cplusplus
	};
#endif

// NOLINTBEGIN(readability-*, bugprone-easily-swappable-parameters, clang-diagnostic-invalid-utf8, clang-diagnostic-invalid-source-encoding, clang-diagnostic-pointer-arith, clang-diagnostic-strict-prototypes, hicpp-uppercase-literal-suffix, cppcoreguidelines-*, performance-*)

/* Setzt eine DATE_AND_TIME-Zeit */
plcdt BrbSetDt(unsigned short nYear, unsigned char nMonth, unsigned char nDay, unsigned char nHour, unsigned char nMinute, unsigned char nSecond)
{
	DTStructure dtStruct;
	DATE_AND_TIME dtTime = BrbSetDtStruct(&dtStruct, nYear, nMonth, nDay, nHour, nMinute, nSecond, 0, 0);
	return dtTime;
}

// NOLINTEND(readability-*, bugprone-easily-swappable-parameters, clang-diagnostic-invalid-utf8, clang-diagnostic-invalid-source-encoding, clang-diagnostic-pointer-arith, clang-diagnostic-strict-prototypes, hicpp-uppercase-literal-suffix, cppcoreguidelines-*, performance-*)
```

#### BrbSetTimespan.c - Setzt eine TIME-Angabe
```c
/********************************************************************
 * COPYRIGHT -- Bernecker + Rainer
 ********************************************************************
 * Library: BrbLib
 * File: BrbSetTimespan.c
 * Author: niedermeierr
 * Created: May 18, 2021
 ********************************************************************
 * Implementation of library BrbLib
 ********************************************************************/

#include <bur/plctypes.h>
#ifdef __cplusplus
	extern "C"
	{
#endif

#include "BrbLib.h"

#ifdef __cplusplus
	};
#endif

// NOLINTBEGIN(readability-*, bugprone-easily-swappable-parameters, clang-diagnostic-invalid-utf8, clang-diagnostic-invalid-source-encoding, clang-diagnostic-pointer-arith, clang-diagnostic-strict-prototypes, hicpp-uppercase-literal-suffix, cppcoreguidelines-*, performance-*)

/* Setzt eine TIME-Zeitspanne */
plctime BrbSetTimespan(signed char nSign, unsigned long nDays, unsigned long nHours, unsigned long nMinutes, unsigned long nSeconds, unsigned long nMilliseconds)
{
	TIME tTime = nBRB_DINT_MAX; // Bei Überschreitung positiven Höchstwert zurückgeben
	UDINT nTime = 0;
	nTime += nMilliseconds;
	nTime += nSeconds * (DINT)nBRB_MILLISECONDS_PER_SECOND;
	nTime += nMinutes * (DINT)nBRB_SECONDS_PER_MINUTE * (DINT)nBRB_MILLISECONDS_PER_SECOND;
	nTime += nHours * (DINT)nBRB_MINUTES_PER_HOUR * (DINT)nBRB_SECONDS_PER_MINUTE * (DINT)nBRB_MILLISECONDS_PER_SECOND;
	nTime += nDays * (DINT)nBRB_HOURS_PER_DAY * (DINT)nBRB_MINUTES_PER_HOUR * (DINT)nBRB_SECONDS_PER_MINUTE * (DINT)nBRB_MILLISECONDS_PER_SECOND;
	if(nSign >= 0)
	{
		if(nTime <= (UDINT)nBRB_DINT_MAX)
		{
			tTime = (DINT)nTime;
		}
	}
	else
	{
		if(nTime <= (UDINT)nBRB_DINT_MAX)
		{
			LREAL rTime = (LREAL)nTime * -1.0;
			tTime = (DINT)rTime;
		}
		else
		{
			tTime = (TIME)(-2147483647 - 1);	// Bei Unterschreitung negativen Höchstwert zurückgeben
		}
	}
	return tTime;
}

// NOLINTEND(readability-*, bugprone-easily-swappable-parameters, clang-diagnostic-invalid-utf8, clang-diagnostic-invalid-source-encoding, clang-diagnostic-pointer-arith, clang-diagnostic-strict-prototypes, hicpp-uppercase-literal-suffix, cppcoreguidelines-*, performance-*)
```

#### BrbSetTimespanT.c - Setzt eine TIME-Angabe per Text
```c
/********************************************************************
 * COPYRIGHT -- Bernecker + Rainer
 ********************************************************************
 * Library: BrbLib
 * File: BrbSetTimespanT.c
 * Author: niedermeierr
 * Created: May 18, 2021
 ********************************************************************
 * Implementation of library BrbLib
 ********************************************************************/

#include <bur/plctypes.h>
#ifdef __cplusplus
	extern "C"
	{
#endif

#include "BrbLib.h"
#include <string.h>

#ifdef __cplusplus
	};
#endif

// NOLINTBEGIN(readability-*, bugprone-easily-swappable-parameters, clang-diagnostic-invalid-utf8, clang-diagnostic-invalid-source-encoding, clang-diagnostic-pointer-arith, clang-diagnostic-strict-prototypes, hicpp-uppercase-literal-suffix, cppcoreguidelines-*, performance-*)

/* Setzt eine TIME-Zeitspanne */
plctime BrbSetTimespanT(plcstring* pTimeText) // NOLINT(readability-function-cognitive-complexity)
{
	TIME tTime = 0;
	if(pTimeText != 0)
	{
		UDINT nTextLen = strlen(pTimeText);
		UDINT nIndex = 0;
		UDINT nIndexStart = 0;
		USINT* pChar = 0;
		SINT nSign = +1;
		STRING sValue[128];
		memset((USINT*)&sValue, 0, sizeof(sValue));
		UDINT nValueLen = 0;
		UDINT nDays = 0;
		UDINT nHours = 0;
		UDINT nMinutes = 0;
		UDINT nSeconds = 0;
		UDINT nMilliseconds = 0;
		if(BrbStringStartsWith(pTimeText, "T#-") == 1)
		{
			nSign = -1;
			nIndexStart += 3;
		}
		else if(BrbStringStartsWith(pTimeText, "T#") == 1)
		{
			nIndexStart += 2;
		}
		else if(BrbStringStartsWith(pTimeText, "-") == 1)
		{
			nSign = -1;
			nIndexStart += 1;
		}
		for(nIndex=nIndexStart; nIndex<nTextLen; nIndex++)
		{
			pChar = (USINT*)(pTimeText + nIndex);
			if(*pChar >= 48 && *pChar <= 57) // 0..9
			{
				sValue[nValueLen] = (char)*pChar;	// Zahl in den Wert übernehmen
				nValueLen += 1;
				sValue[nValueLen] = 0; // Nullterminierung
			}
			else if(*pChar == 100) // d
			{
				if(nValueLen > 0)
				{
					nDays = BrbAsciiToUdint(sValue);
					memset((USINT*)&sValue, 0, sizeof(sValue));
					nValueLen = 0;
				}
			}
			else if(*pChar == 104) // h
			{
				if(nValueLen > 0)
				{
					nHours = BrbAsciiToUdint(sValue);
					memset((USINT*)&sValue, 0, sizeof(sValue));
					nValueLen = 0;
				}
			}
			else if(*pChar == 109 && *(pChar+1) != 115) // m
			{
				if(nValueLen > 0)
				{
					nMinutes = BrbAsciiToUdint(sValue);
					memset((USINT*)&sValue, 0, sizeof(sValue));
					nValueLen = 0;
				}
			}
			else if(*pChar == 115 && (nIndex == 0 || *(pChar-1) != 109)) // s
			{
				if(nValueLen > 0)
				{
					nSeconds = BrbAsciiToUdint(sValue);
					memset((USINT*)&sValue, 0, sizeof(sValue));
					nValueLen = 0;
				}
			}
			else if(*pChar == 109 && *(pChar+1) == 115) // ms
			{
				if(nValueLen > 0)
				{
					nMilliseconds = BrbAsciiToUdint(sValue);
					memset((USINT*)&sValue, 0, sizeof(sValue));
					nValueLen = 0;
					nIndex++; // nächstes 's' überspringen
				}
			}
		}
		tTime = BrbSetTimespan(nSign, nDays, nHours, nMinutes, nSeconds, nMilliseconds);
	}
	return tTime;
}

// NOLINTEND(readability-*, bugprone-easily-swappable-parameters, clang-diagnostic-invalid-utf8, clang-diagnostic-invalid-source-encoding, clang-diagnostic-pointer-arith, clang-diagnostic-strict-prototypes, hicpp-uppercase-literal-suffix, cppcoreguidelines-*, performance-*)
```

#### BrbGetTimeText.c - Gibt die angegebene Zeit als Text zurück yyyy.MM.dd hh:mm:ss:mil
```c
/********************************************************************
 * COPYRIGHT -- Bernecker + Rainer
 ********************************************************************
 * Library: BrbLib
 * File: BrbGetTimeText.c
 * Author: niedermeierr
 * Created: June 11, 2013
 ********************************************************************
 * Implementation of library BrbLib
 ********************************************************************/

#include <bur/plctypes.h>
#ifdef __cplusplus
	extern "C"
	{
#endif

#include "BrbLib.h"
#include <string.h>

#ifdef __cplusplus
	};
#endif

// NOLINTBEGIN(readability-*, bugprone-easily-swappable-parameters, clang-diagnostic-invalid-utf8, clang-diagnostic-invalid-source-encoding, clang-diagnostic-pointer-arith, clang-diagnostic-strict-prototypes, hicpp-uppercase-literal-suffix, cppcoreguidelines-*, performance-*)

/* Gibt die angegebene RTC-Zeit als Text zurück */
unsigned short BrbGetTimeText(struct RTCtime_typ* pTime, plcstring* pText, unsigned long nTextSize, plcstring* pFormat) // NOLINT(readability-function-cognitive-complexity)
{
	// Prüfung der Parameter
	if(pTime == 0)
	{
		return eBRB_ERR_NULL_POINTER;
	}
	if(pText == 0)
	{
		return eBRB_ERR_NULL_POINTER;
	}
	if(nTextSize == 0)
	{
		return eBRB_ERR_INVALID_PARAMETER;
	}
	if(pFormat == 0)
	{
		return eBRB_ERR_NULL_POINTER;
	}
	// Alle Stellen werden mit führenden Nullen aufgefüllt
	BrbStringCopy(pText, pFormat, nTextSize);
	STRING sItoA[20];
	memset((USINT*)sItoA, 0, sizeof(sItoA));
	if(BrbStringGetAdrOf(pText, "yyyy", 0) != 0)
	{
		brsitoa((DINT)pTime->year, (UDINT)&sItoA);
		BrbStringPadLeft(sItoA, "0", 4);
		BrbStringReplace(pText, "yyyy", sItoA);
	}
	else if(BrbStringGetAdrOf(pText, "yy", 0) != 0)
	{
		pTime->year -= 2000;
		brsitoa((DINT)pTime->year, (UDINT)&sItoA);
		BrbStringPadLeft(sItoA, "0", 2);
		BrbStringReplace(pText, "yy", sItoA);
	}
	if(BrbStringGetAdrOf(pText, "mil", 0) != 0)
	{
		brsitoa((DINT)pTime->millisec, (UDINT)&sItoA);
		if(pTime->millisec < 10)
		{
			BrbStringInsert(sItoA, 0, "00");
		}
		else if(pTime->millisec < 100)
		{
			BrbStringInsert(sItoA, 0, "0");
		}
		BrbStringReplace(pText, "mil", sItoA);
	}
	if(BrbStringGetAdrOf(pText, "mic", 0) != 0)
	{
		brsitoa((DINT)pTime->microsec, (UDINT)&sItoA);
		if(pTime->microsec < 10)
		{
			BrbStringInsert(sItoA, 0, "00");
		}
		else if(pTime->microsec < 100)
		{
			BrbStringInsert(sItoA, 0, "0");
		}
		BrbStringReplace(pText, "mic", sItoA);
	}
	if(BrbStringGetAdrOf(pText, "mm", 0) != 0)
	{
		brsitoa((DINT)pTime->month, (UDINT)&sItoA);
		if(pTime->month < 10)
		{
			BrbStringInsert(sItoA, 0, "0");
		}
		BrbStringReplace(pText, "mm", sItoA);
	}
	else if(BrbStringGetAdrOf(pText, "m", 0) != 0)
	{
		brsitoa((DINT)pTime->month, (UDINT)&sItoA);
		BrbStringReplace(pText, "m", sItoA);
	}
	if(BrbStringGetAdrOf(pText, "dd", 0) != 0)
	{
		brsitoa((DINT)pTime->day, (UDINT)&sItoA);
		if(pTime->day < 10)
		{
			BrbStringInsert(sItoA, 0, "0");
		}
		BrbStringReplace(pText, "dd", sItoA);
	}
	else if(BrbStringGetAdrOf(pText, "d", 0) != 0)
	{
		brsitoa((DINT)pTime->day, (UDINT)&sItoA);
		BrbStringReplace(pText, "d", sItoA);
	}
	if(BrbStringGetAdrOf(pText, "hh", 0) != 0)
	{
		brsitoa((DINT)pTime->hour, (UDINT)&sItoA);
		if(pTime->hour < 10)
		{
			BrbStringInsert(sItoA, 0, "0");
		}
		BrbStringReplace(pText, "hh", sItoA);
	}
	else if(BrbStringGetAdrOf(pText, "h", 0) != 0)
	{
		brsitoa((DINT)pTime->hour, (UDINT)&sItoA);
		BrbStringReplace(pText, "h", sItoA);
	}
	if(BrbStringGetAdrOf(pText, "MM", 0) != 0)
	{
		brsitoa((DINT)pTime->minute, (UDINT)&sItoA);
		if(pTime->minute < 10)
		{
			BrbStringInsert(sItoA, 0, "0");
		}
		BrbStringReplace(pText, "MM", sItoA);
	}
	else if(BrbStringGetAdrOf(pText, "M", 0) != 0)
	{
		brsitoa((DINT)pTime->minute, (UDINT)&sItoA);
		BrbStringReplace(pText, "M", sItoA);
	}
	if(BrbStringGetAdrOf(pText, "ss", 0) != 0)
	{
		brsitoa((DINT)pTime->second, (UDINT)&sItoA);
		if(pTime->second < 10)
		{
			BrbStringInsert(sItoA, 0, "0");
		}
		BrbStringReplace(pText, "ss", sItoA);
	}
	else if(BrbStringGetAdrOf(pText, "s", 0) != 0)
	{
		brsitoa((DINT)pTime->second, (UDINT)&sItoA);
		BrbStringReplace(pText, "s", sItoA);
	}
	return eBRB_ERR_OK;
}

// NOLINTEND(readability-*, bugprone-easily-swappable-parameters, clang-diagnostic-invalid-utf8, clang-diagnostic-invalid-source-encoding, clang-diagnostic-pointer-arith, clang-diagnostic-strict-prototypes, hicpp-uppercase-literal-suffix, cppcoreguidelines-*, performance-*)
```

#### BrbGetCurrentTimeText.c - Gibt die aktuelle Zeit als Text zurück: yyyy.MM.dd hh:mm:ss:mil
```c
/********************************************************************
 * COPYRIGHT -- Bernecker + Rainer
 ********************************************************************
 * Library: BrbLib
 * File: BrbGetCurrentTimeText.c
 * Author: niedermeierr
 * Created: June 11, 2013
 ********************************************************************
 * Implementation of library BrbLib
 ********************************************************************/

#include <bur/plctypes.h>
#ifdef __cplusplus
	extern "C"
	{
#endif

#include "BrbLib.h"

#ifdef __cplusplus
	};
#endif

// NOLINTBEGIN(readability-*, bugprone-easily-swappable-parameters, clang-diagnostic-invalid-utf8, clang-diagnostic-invalid-source-encoding, clang-diagnostic-pointer-arith, clang-diagnostic-strict-prototypes, hicpp-uppercase-literal-suffix, cppcoreguidelines-*, performance-*)

/* Gibt die aktuelle Zeit als Text zurück */
unsigned short BrbGetCurrentTimeText(plcstring* pText, unsigned long nTextSize, plcstring* pFormat)
{
	RTCtime_typ Time;
	RTC_gettime(&Time);
	return BrbGetTimeText(&Time, pText, nTextSize, pFormat);
}

// NOLINTEND(readability-*, bugprone-easily-swappable-parameters, clang-diagnostic-invalid-utf8, clang-diagnostic-invalid-source-encoding, clang-diagnostic-pointer-arith, clang-diagnostic-strict-prototypes, hicpp-uppercase-literal-suffix, cppcoreguidelines-*, performance-*)
```

#### BrbGetTimeTextDtStruct.c - Gibt die angegebene Zeit als Text zurück yyyy.MM.dd hh:mm:ss:mil
```c
/********************************************************************
 * COPYRIGHT -- Bernecker + Rainer
 ********************************************************************
 * Library: BrbLib
 * File: BrbGetTimeTextDtStruct.c
 * Author: niedermeierr
 * Created: June 11, 2013
 ********************************************************************
 * Implementation of library BrbLib
 ********************************************************************/

#include <bur/plctypes.h>
#ifdef __cplusplus
	extern "C"
	{
#endif

#include "BrbLib.h"

#ifdef __cplusplus
	};
#endif

// NOLINTBEGIN(readability-*, bugprone-easily-swappable-parameters, clang-diagnostic-invalid-utf8, clang-diagnostic-invalid-source-encoding, clang-diagnostic-pointer-arith, clang-diagnostic-strict-prototypes, hicpp-uppercase-literal-suffix, cppcoreguidelines-*, performance-*)

/* Gibt die angegebene DtStruct-Zeit als Text zurück */
unsigned short BrbGetTimeTextDtStruct(struct DTStructure* pTime, plcstring* pText, unsigned long nTextSize, plcstring* pFormat)
{
	// Prüfung der Parameter
	if(pTime == 0)
	{
		return eBRB_ERR_NULL_POINTER;
	}
	if(pText == 0)
	{
		return eBRB_ERR_NULL_POINTER;
	}
	if(nTextSize == 0)
	{
		return eBRB_ERR_INVALID_PARAMETER;
	}
	if(pFormat == 0)
	{
		return eBRB_ERR_NULL_POINTER;
	}
	// Text ermitteln
	RTCtime_typ RtcTime;
	RtcTime.year = pTime->year;
	RtcTime.month = pTime->month;
	RtcTime.day = pTime->day;
	RtcTime.hour = pTime->hour;
	RtcTime.minute = pTime->minute;
	RtcTime.second = pTime->second;
	RtcTime.millisec = pTime->millisec;
	RtcTime.microsec = pTime->microsec;
	return BrbGetTimeText(&RtcTime, pText, nTextSize, pFormat);
}

// NOLINTEND(readability-*, bugprone-easily-swappable-parameters, clang-diagnostic-invalid-utf8, clang-diagnostic-invalid-source-encoding, clang-diagnostic-pointer-arith, clang-diagnostic-strict-prototypes, hicpp-uppercase-literal-suffix, cppcoreguidelines-*, performance-*)
```

#### BrbGetTimeTextDt.c - Gibt die angegebene Zeit als Text zurück yyyy.MM.dd hh.mm.ss
```c
/********************************************************************
 * COPYRIGHT -- Bernecker + Rainer
 ********************************************************************
 * Library: BrbLib
 * File: BrbGetTimeTextDt.c
 * Author: niedermeierr
 * Created: June 11, 2013
 ********************************************************************
 * Implementation of library BrbLib
 ********************************************************************/

#include <bur/plctypes.h>
#ifdef __cplusplus
	extern "C"
	{
#endif

#include "BrbLib.h"

#ifdef __cplusplus
	};
#endif

// NOLINTBEGIN(readability-*, bugprone-easily-swappable-parameters, clang-diagnostic-invalid-utf8, clang-diagnostic-invalid-source-encoding, clang-diagnostic-pointer-arith, clang-diagnostic-strict-prototypes, hicpp-uppercase-literal-suffix, cppcoreguidelines-*, performance-*)

/* Gibt die angegebene DT-Zeit als Text zurück */
unsigned short BrbGetTimeTextDt(plcdt dtTime, plcstring* pText, unsigned long nTextSize, plcstring* pFormat)
{
	if(pText == 0)
	{
		return eBRB_ERR_NULL_POINTER;
	}
	if(nTextSize == 0)
	{
		return eBRB_ERR_INVALID_PARAMETER;
	}
	if(pFormat == 0)
	{
		return eBRB_ERR_NULL_POINTER;
	}
	// Text ermitteln
	DTStructure DtStruct;
	DT_TO_DTStructure(dtTime, (UDINT)&DtStruct);
	return BrbGetTimeTextDtStruct(&DtStruct, pText, nTextSize, pFormat);
}

// NOLINTEND(readability-*, bugprone-easily-swappable-parameters, clang-diagnostic-invalid-utf8, clang-diagnostic-invalid-source-encoding, clang-diagnostic-pointer-arith, clang-diagnostic-strict-prototypes, hicpp-uppercase-literal-suffix, cppcoreguidelines-*, performance-*)
```

#### BrbGetDtFromTimeText.c - Wandelt einen Zeit-Text in eine Zeit-Struktur um
```c
/********************************************************************
 * COPYRIGHT -- Bernecker + Rainer
 ********************************************************************
 * Library: BrbLib
 * File: BrbGetDtFromTimeText.c
 * Author: niedermeierr
 * Created: June 25, 2013
 ********************************************************************
 * Implementation of library BrbLib
 ********************************************************************/

#include <bur/plctypes.h>
#ifdef __cplusplus
	extern "C"
	{
#endif

#include "BrbLib.h"
#include <string.h>

#ifdef __cplusplus
	};
#endif

// NOLINTBEGIN(readability-*, bugprone-easily-swappable-parameters, clang-diagnostic-invalid-utf8, clang-diagnostic-invalid-source-encoding, clang-diagnostic-pointer-arith, clang-diagnostic-strict-prototypes, hicpp-uppercase-literal-suffix, cppcoreguidelines-*, performance-*)

/* Wandelt einen Zeit-Text in eine Zeit um */
plcdt BrbGetDtFromTimeText(plcstring* pTimeText, plcstring* pFormat) // NOLINT(readability-function-cognitive-complexity)
{
	if(pTimeText == 0)
	{
		return 0;
	}
	if(pFormat == 0)
	{
		return 0;
	}
	DATE_AND_TIME dtResult = 0;
	UDINT nTimeTextLen = strlen(pTimeText);
	UDINT nFormatLen = strlen(pFormat);
	if(nTimeTextLen >= nFormatLen)
	{
		UDINT nAdr = 0;
		UDINT nOffset = 0;
		STRING sValue[20];
		DTStructure DtStruct;
		memset((USINT*)&DtStruct, 0, sizeof(DtStruct));
		nAdr = (UDINT)BrbStringGetAdrOf(pFormat, "yyyy", nFormatLen); // NOLINT(clang-diagnostic-bad-function-cast)
		if(nAdr >= (UDINT)pFormat)
		{
			nOffset = nAdr - (UDINT)pFormat;
			BrbStringGetSubText(pTimeText, nOffset, 4, sValue);
			DtStruct.year = (UINT)brsatoi((UDINT)&sValue);
		}
		else
		{
			nAdr = (UDINT)BrbStringGetAdrOf(pFormat, "yy", nFormatLen); // NOLINT(clang-diagnostic-bad-function-cast)
			if(nAdr >= (UDINT)pFormat)
			{
				nOffset = nAdr - (UDINT)pFormat;
				BrbStringGetSubText(pTimeText, nOffset, 2, sValue);
				DtStruct.year = (UINT)brsatoi((UDINT)&sValue) + 2000;
			}
		}
		nAdr = (UDINT)BrbStringGetAdrOf(pFormat, "mm", nFormatLen); // NOLINT(clang-diagnostic-bad-function-cast)
		if(nAdr >= (UDINT)pFormat)
		{
			nOffset = nAdr - (UDINT)pFormat;
			BrbStringGetSubText(pTimeText, nOffset, 2, sValue);
			DtStruct.month = (USINT)brsatoi((UDINT)&sValue);
		}
		else
		{
			nAdr = (UDINT)BrbStringGetAdrOf(pFormat, "m", nFormatLen); // NOLINT(clang-diagnostic-bad-function-cast)
			if(nAdr >= (UDINT)pFormat)
			{
				nOffset = nAdr - (UDINT)pFormat;
				BrbStringGetSubText(pTimeText, nOffset, 1, sValue);
				DtStruct.month = (USINT)brsatoi((UDINT)&sValue);
			}
		}
		nAdr = (UDINT)BrbStringGetAdrOf(pFormat, "dd", nFormatLen); // NOLINT(clang-diagnostic-bad-function-cast)
		if(nAdr >= (UDINT)pFormat)
		{
			nOffset = nAdr - (UDINT)pFormat;
			BrbStringGetSubText(pTimeText, nOffset, 2, sValue);
			DtStruct.day = (USINT)brsatoi((UDINT)&sValue);
		}
		else
		{
			nAdr = (UDINT)BrbStringGetAdrOf(pFormat, "d", nFormatLen); // NOLINT(clang-diagnostic-bad-function-cast)
			if(nAdr >= (UDINT)pFormat)
			{
				nOffset = nAdr - (UDINT)pFormat;
				BrbStringGetSubText(pTimeText, nOffset, 1, sValue);
				DtStruct.day = (USINT)brsatoi((UDINT)&sValue);
			}
		}
		nAdr = (UDINT)BrbStringGetAdrOf(pFormat, "hh", nFormatLen); // NOLINT(clang-diagnostic-bad-function-cast)
		if(nAdr >= (UDINT)pFormat)
		{
			nOffset = nAdr - (UDINT)pFormat;
			BrbStringGetSubText(pTimeText, nOffset, 2, sValue);
			DtStruct.hour = (USINT)brsatoi((UDINT)&sValue);
		}
		else
		{
			nAdr = (UDINT)BrbStringGetAdrOf(pFormat, "h", nFormatLen); // NOLINT(clang-diagnostic-bad-function-cast)
			if(nAdr >= (UDINT)pFormat)
			{
				nOffset = nAdr - (UDINT)pFormat;
				BrbStringGetSubText(pTimeText, nOffset, 1, sValue);
				DtStruct.hour = (USINT)brsatoi((UDINT)&sValue);
			}
		}
		nAdr = (UDINT)BrbStringGetAdrOf(pFormat, "MM", nFormatLen); // NOLINT(clang-diagnostic-bad-function-cast)
		if(nAdr >= (UDINT)pFormat)
		{
			nOffset = nAdr - (UDINT)pFormat;
			BrbStringGetSubText(pTimeText, nOffset, 2, sValue);
			DtStruct.minute = (USINT)brsatoi((UDINT)&sValue);
		}
		else
		{
			nAdr = (UDINT)BrbStringGetAdrOf(pFormat, "M", nFormatLen); // NOLINT(clang-diagnostic-bad-function-cast)
			if(nAdr >= (UDINT)pFormat)
			{
				nOffset = nAdr - (UDINT)pFormat;
				BrbStringGetSubText(pTimeText, nOffset, 1, sValue);
				DtStruct.minute = (USINT)brsatoi((UDINT)&sValue);
			}
		}
		nAdr = (UDINT)BrbStringGetAdrOf(pFormat, "ss", nFormatLen); // NOLINT(clang-diagnostic-bad-function-cast)
		if(nAdr >= (UDINT)pFormat)
		{
			nOffset = nAdr - (UDINT)pFormat;
			BrbStringGetSubText(pTimeText, nOffset, 2, sValue);
			DtStruct.second = (USINT)brsatoi((UDINT)&sValue);
		}
		else
		{
			nAdr = (UDINT)BrbStringGetAdrOf(pFormat, "s", nFormatLen); // NOLINT(clang-diagnostic-bad-function-cast)
			if(nAdr >= (UDINT)pFormat)
			{
				nOffset = nAdr - (UDINT)pFormat;
				BrbStringGetSubText(pTimeText, nOffset, 1, sValue);
				DtStruct.second = (USINT)brsatoi((UDINT)&sValue);
			}
		}
		nAdr = (UDINT)BrbStringGetAdrOf(pFormat, "mil", nFormatLen); // NOLINT(clang-diagnostic-bad-function-cast)
		if(nAdr >= (UDINT)pFormat)
		{
			nOffset = nAdr - (UDINT)pFormat;
			BrbStringGetSubText(pTimeText, nOffset, 3, sValue);
			DtStruct.millisec = (UINT)brsatoi((UDINT)&sValue);
		}
		nAdr = (UDINT)BrbStringGetAdrOf(pFormat, "mic", nFormatLen); // NOLINT(clang-diagnostic-bad-function-cast)
		if(nAdr >= (UDINT)pFormat)
		{
			nOffset = nAdr - (UDINT)pFormat;
			BrbStringGetSubText(pTimeText, nOffset, 3, sValue);
			DtStruct.microsec = (UINT)brsatoi((UDINT)&sValue);
		}
		dtResult = DTStructure_TO_DT((UDINT)&DtStruct);
	}
	return dtResult;
}

// NOLINTEND(readability-*, bugprone-easily-swappable-parameters, clang-diagnostic-invalid-utf8, clang-diagnostic-invalid-source-encoding, clang-diagnostic-pointer-arith, clang-diagnostic-strict-prototypes, hicpp-uppercase-literal-suffix, cppcoreguidelines-*, performance-*)
```

#### BrbRtcTimeToDtStruct.c - Wandelt eine RTC-Zeit in eine DtStruct-Zeit
```c
/********************************************************************
 * COPYRIGHT -- Bernecker + Rainer
 ********************************************************************
 * Library: BrbLib
 * File: BrbRtcTimeToDtStruct.c
 * Author: niedermeierr
 * Created: June 25, 2013
 ********************************************************************
 * Implementation of library BrbLib
 ********************************************************************/

#include <bur/plctypes.h>
#ifdef __cplusplus
	extern "C"
	{
#endif

#include "BrbLib.h"

#ifdef __cplusplus
	};
#endif

// NOLINTBEGIN(readability-*, bugprone-easily-swappable-parameters, clang-diagnostic-invalid-utf8, clang-diagnostic-invalid-source-encoding, clang-diagnostic-pointer-arith, clang-diagnostic-strict-prototypes, hicpp-uppercase-literal-suffix, cppcoreguidelines-*, performance-*)

/* Wandelt eine RTC-Zeit in eine DtStruct-Zeit */
unsigned short BrbRtcTimeToDtStruct(struct RTCtime_typ* pRtcTime, struct DTStructure* pDtStruct)
{
	// Prüfung der Parameter
	if(pRtcTime == 0)
	{
		return eBRB_ERR_NULL_POINTER;
	}
	if(pDtStruct == 0)
	{
		return eBRB_ERR_NULL_POINTER;
	}
	// Wandlung
	pDtStruct->year = pRtcTime->year;
	pDtStruct->month = pRtcTime->month;
	pDtStruct->day = pRtcTime->day;
	pDtStruct->wday = 0;
	pDtStruct->hour = pRtcTime->hour;
	pDtStruct->minute = pRtcTime->minute;
	pDtStruct->second = pRtcTime->second;
	pDtStruct->millisec = pRtcTime->millisec;
	pDtStruct->microsec = pRtcTime->microsec;
	return eBRB_ERR_OK;
}

// NOLINTEND(readability-*, bugprone-easily-swappable-parameters, clang-diagnostic-invalid-utf8, clang-diagnostic-invalid-source-encoding, clang-diagnostic-pointer-arith, clang-diagnostic-strict-prototypes, hicpp-uppercase-literal-suffix, cppcoreguidelines-*, performance-*)
```
